Universal Robots URScript: infinity_multi.urscript

# UR10 -- infinity_multi
# Points: 3200   v=2.0 rad/s   a=1.7 rad/s2
# Generated by send_xyz.py
def run_infinity_multi():
  set_tool_voltage(12)           # power tool connector (12V for LED)
  set_tool_digital_out(0, False) # LED off initially
  movej([1.57, -1.2, 1.6, -0.4, 1.57, 0.0], a=0.4, v=0.2)   # go to home first
  movej([2.38, -1.326, 1.6, -0.4, 1.57, 0.0], a=0.4, v=0.2)   # move to pattern start
  sleep(1.5)   # pause — home ≠ start (dist=0.820 rad)
  set_tool_digital_out(0, True)  # LED on — drawing starts
  movej([2.38, -1.3359, 1.6, -0.4, 1.57, 0.0], a=1.7, v=2.0, r=0.08)
  movej([2.3799, -1.3458, 1.6, -0.4, 1.57, 0.0], a=1.7, v=2.0, r=0.08)
  movej([2.3798, -1.3557, 1.6, -0.4, 1.57, 0.0], a=1.7, v=2.0, r=0.08)
  movej([2.3796, -1.3656, 1.6, -0.4, 1.57, 0.0], a=1.7, v=2.0, r=0.08)
  movej([2.3794, -1.3755, 1.6, -0.4, 1.57, 0.0], a=1.7, v=2.0, r=0.08)
  movej([2.3791, -1.3854, 1.6, -0.4, 1.57, 0.0], a=1.7, v=2.0, r=0.08)
  movej([2.3788, -1.3952, 1.6, -0.4, 1.57, 0.0], a=1.7, v=2.0, r=0.08)
  movej([2.3784, -1.4051, 1.6, -0.4, 1.57, 0.0], a=1.7, v=2.0, r=0.08)
  movej([2.378, -1.4149, 1.6, -0.4, 1.57, 0.0], a=1.7, v=2.0, r=0.08)
  movej([2.3775, -1.4247, 1.6, -0.4, 1.57, 0.0], a=1.7, v=2.0, r=0.08)
  movej([2.377, -1.4344, 1.6, -0.4, 1.57, 0.0], a=1.7, v=2.0, r=0.08)
  movej([2.3764, -1.4442, 1.6, -0.4, 1.57, 0.0], a=1.7, v=2.0, r=0.08)
  movej([2.3758, -1.4539, 1.6, -0.4, 1.57, 0.0], a=1.7, v=2.0, r=0.08)
  movej([2.3751, -1.4636, 1.6, -0.4, 1.57, 0.0], a=1.7, v=2.0, r=0.08)
  movej([2.3744, -1.4733, 1.6, -0.4, 1.57, 0.0], a=1.7, v=2.0, r=0.08)
  movej([2.3736, -1.4829, 1.6, -0.4, 1.57, 0.0], a=1.7, v=2.0, r=0.08)
  movej([2.3728, -1.4924, 1.6, -0.4, 1.57, 0.0], a=1.7, v=2.0, r=0.08)
  movej([2.3719, -1.502, 1.6, -0.4, 1.57, 0.0], a=1.7, v=2.0, r=0.08)
  movej([2.371, -1.5115, 1.6, -0.4, 1.57, 0.0], a=1.7, v=2.0, r=0.08)
  movej([2.37, -1.5209, 1.6, -0.4, 1.57, 0.0], a=1.7, v=2.0, r=0.08)
  movej([2.369, -1.5303, 1.6, -0.4, 1.57, 0.0], a=1.7, v=2.0, r=0.08)
  movej([2.3679, -1.5397, 1.6, -0.4, 1.57, 0.0], a=1.7, v=2.0, r=0.08)
  movej([2.3668, -1.549, 1.6, -0.4, 1.57, 0.0], a=1.7, v=2.0, r=0.08)
  movej([2.3656, -1.5582, 1.6, -0.4, 1.57, 0.0], a=1.7, v=2.0, r=0.08)
  movej([2.3644, -1.5674, 1.6, -0.4, 1.57, 0.0], a=1.7, v=2.0, r=0.08)
  movej([2.3631, -1.5765, 1.6, -0.4, 1.57, 0.0], a=1.7, v=2.0, r=0.08)
  movej([2.3618, -1.5856, 1.6, -0.4, 1.57, 0.0], a=1.7, v=2.0, r=0.08)
  movej([2.3604, -1.5946, 1.6, -0.4, 1.57, 0.0], a=1.7, v=2.0, r=0.08)
  movej([2.359, -1.6035, 1.6, -0.4, 1.57, 0.0], a=1.7, v=2.0, r=0.08)
  movej([2.3576, -1.6123, 1.6, -0.4, 1.57, 0.0], a=1.7, v=2.0, r=0.08)
  movej([2.3561, -1.6211, 1.6, -0.4, 1.57, 0.0], a=1.7, v=2.0, r=0.08)
  movej([2.3545, -1.6299, 1.6, -0.4, 1.57, 0.0], a=1.7, v=2.0, r=0.08)
  movej([2.3529, -1.6385, 1.6, -0.4, 1.57, 0.0], a=1.7, v=2.0, r=0.08)
  movej([2.3512, -1.6471, 1.6, -0.4, 1.57, 0.0], a=1.7, v=2.0, r=0.08)
  movej([2.3495, -1.6555, 1.6, -0.4, 1.57, 0.0], a=1.7, v=2.0, r=0.08)
  movej([2.3478, -1.6639, 1.6, -0.4, 1.57, 0.0], a=1.7, v=2.0, r=0.08)
  movej([2.346, -1.6723, 1.6, -0.4, 1.57, 0.0], a=1.7, v=2.0, r=0.08)
  movej([2.3441, -1.6805, 1.6, -0.4, 1.57, 0.0], a=1.7, v=2.0, r=0.08)
  movej([2.3422, -1.6886, 1.6, -0.4, 1.57, 0.0], a=1.7, v=2.0, r=0.08)
  movej([2.3403, -1.6967, 1.6, -0.4, 1.57, 0.0], a=1.7, v=2.0, r=0.08)
  movej([2.3383, -1.7047, 1.6, -0.4, 1.57, 0.0], a=1.7, v=2.0, r=0.08)
  movej([2.3362, -1.7125, 1.6, -0.4, 1.57, 0.0], a=1.7, v=2.0, r=0.08)
  movej([2.3341, -1.7203, 1.6, -0.4, 1.57, 0.0], a=1.7, v=2.0, r=0.08)
  movej([2.332, -1.728, 1.6, -0.4, 1.57, 0.0], a=1.7, v=2.0, r=0.08)
  movej([2.3298, -1.7356, 1.6, -0.4, 1.57, 0.0], a=1.7, v=2.0, r=0.08)
  movej([2.3276, -1.7431, 1.6, -0.4, 1.57, 0.0], a=1.7, v=2.0, r=0.08)
  movej([2.3253, -1.7504, 1.6, -0.4, 1.57, 0.0], a=1.7, v=2.0, r=0.08)
  movej([2.323, -1.7577, 1.6, -0.4, 1.57, 0.0], a=1.7, v=2.0, r=0.08)
  movej([2.3206, -1.7649, 1.6, -0.4, 1.57, 0.0], a=1.7, v=2.0, r=0.08)
  movej([2.3182, -1.7719, 1.6, -0.4, 1.57, 0.0], a=1.7, v=2.0, r=0.08)
  movej([2.3157, -1.7789, 1.6, -0.4, 1.57, 0.0], a=1.7, v=2.0, r=0.08)
  movej([2.3132, -1.7857, 1.6, -0.4, 1.57, 0.0], a=1.7, v=2.0, r=0.08)
  movej([2.3107, -1.7924, 1.6, -0.4, 1.57, 0.0], a=1.7, v=2.0, r=0.08)
  movej([2.3081, -1.799, 1.6, -0.4, 1.57, 0.0], a=1.7, v=2.0, r=0.08)
  movej([2.3054, -1.8055, 1.6, -0.4, 1.57, 0.0], a=1.7, v=2.0, r=0.08)
  movej([2.3027, -1.8119, 1.6, -0.4, 1.57, 0.0], a=1.7, v=2.0, r=0.08)
  movej([2.3, -1.8181, 1.6, -0.4, 1.57, 0.0], a=1.7, v=2.0, r=0.08)
  movej([2.2972, -1.8242, 1.6, -0.4, 1.57, 0.0], a=1.7, v=2.0, r=0.08)
  movej([2.2944, -1.8302, 1.6, -0.4, 1.57, 0.0], a=1.7, v=2.0, r=0.08)
  movej([2.2915, -1.8361, 1.6, -0.4, 1.57, 0.0], a=1.7, v=2.0, r=0.08)
  movej([2.2886, -1.8419, 1.6, -0.4, 1.57, 0.0], a=1.7, v=2.0, r=0.08)
  movej([2.2856, -1.8475, 1.6, -0.4, 1.57, 0.0], a=1.7, v=2.0, r=0.08)
  movej([2.2826, -1.853, 1.6, -0.4, 1.57, 0.0], a=1.7, v=2.0, r=0.08)
  movej([2.2796, -1.8584, 1.6, -0.4, 1.57, 0.0], a=1.7, v=2.0, r=0.08)
  movej([2.2765, -1.8636, 1.6, -0.4, 1.57, 0.0], a=1.7, v=2.0, r=0.08)
  movej([2.2733, -1.8687, 1.6, -0.4, 1.57, 0.0], a=1.7, v=2.0, r=0.08)
  movej([2.2701, -1.8736, 1.6, -0.4, 1.57, 0.0], a=1.7, v=2.0, r=0.08)
  movej([2.2669, -1.8785, 1.6, -0.4, 1.57, 0.0], a=1.7, v=2.0, r=0.08)
  movej([2.2637, -1.8832, 1.6, -0.4, 1.57, 0.0], a=1.7, v=2.0, r=0.08)
  movej([2.2603, -1.8877, 1.6, -0.4, 1.57, 0.0], a=1.7, v=2.0, r=0.08)
  movej([2.257, -1.8921, 1.6, -0.4, 1.57, 0.0], a=1.7, v=2.0, r=0.08)
  movej([2.2536, -1.8964, 1.6, -0.4, 1.57, 0.0], a=1.7, v=2.0, r=0.08)
  movej([2.2502, -1.9006, 1.6, -0.4, 1.57, 0.0], a=1.7, v=2.0, r=0.08)
  movej([2.2467, -1.9045, 1.6, -0.4, 1.57, 0.0], a=1.7, v=2.0, r=0.08)
  movej([2.2432, -1.9084, 1.6, -0.4, 1.57, 0.0], a=1.7, v=2.0, r=0.08)
  movej([2.2396, -1.9121, 1.6, -0.4, 1.57, 0.0], a=1.7, v=2.0, r=0.08)
  movej([2.236, -1.9157, 1.6, -0.4, 1.57, 0.0], a=1.7, v=2.0, r=0.08)
  movej([2.2323, -1.9191, 1.6, -0.4, 1.57, 0.0], a=1.7, v=2.0, r=0.08)
  movej([2.2287, -1.9224, 1.6, -0.4, 1.57, 0.0], a=1.7, v=2.0, r=0.08)
  movej([2.2249, -1.9255, 1.6, -0.4, 1.57, 0.0], a=1.7, v=2.0, r=0.08)
  movej([2.2212, -1.9284, 1.6, -0.4, 1.57, 0.0], a=1.7, v=2.0, r=0.08)
  movej([2.2174, -1.9313, 1.6, -0.4, 1.57, 0.0], a=1.7, v=2.0, r=0.08)
  movej([2.2135, -1.9339, 1.6, -0.4, 1.57, 0.0], a=1.7, v=2.0, r=0.08)
  movej([2.2096, -1.9365, 1.6, -0.4, 1.57, 0.0], a=1.7, v=2.0, r=0.08)
  movej([2.2057, -1.9388, 1.6, -0.4, 1.57, 0.0], a=1.7, v=2.0, r=0.08)
  movej([2.2017, -1.9411, 1.6, -0.4, 1.57, 0.0], a=1.7, v=2.0, r=0.08)
  movej([2.1977, -1.9431, 1.6, -0.4, 1.57, 0.0], a=1.7, v=2.0, r=0.08)
  movej([2.1937, -1.945, 1.6, -0.4, 1.57, 0.0], a=1.7, v=2.0, r=0.08)
  movej([2.1896, -1.9468, 1.6, -0.4, 1.57, 0.0], a=1.7, v=2.0, r=0.08)
  movej([2.1855, -1.9484, 1.6, -0.4, 1.57, 0.0], a=1.7, v=2.0, r=0.08)
  movej([2.1813, -1.9499, 1.6, -0.4, 1.57, 0.0], a=1.7, v=2.0, r=0.08)
  movej([2.1771, -1.9512, 1.6, -0.4, 1.57, 0.0], a=1.7, v=2.0, r=0.08)
  movej([2.1729, -1.9523, 1.6, -0.4, 1.57, 0.0], a=1.7, v=2.0, r=0.08)
  movej([2.1686, -1.9533, 1.6, -0.4, 1.57, 0.0], a=1.7, v=2.0, r=0.08)
  movej([2.1643, -1.9542, 1.6, -0.4, 1.57, 0.0], a=1.7, v=2.0, r=0.08)
  movej([2.1599, -1.9548, 1.6, -0.4, 1.57, 0.0], a=1.7, v=2.0, r=0.08)
  movej([2.1556, -1.9554, 1.6, -0.4, 1.57, 0.0], a=1.7, v=2.0, r=0.08)
  movej([2.1511, -1.9557, 1.6, -0.4, 1.57, 0.0], a=1.7, v=2.0, r=0.08)
  movej([2.1467, -1.9559, 1.6, -0.4, 1.57, 0.0], a=1.7, v=2.0, r=0.08)
  movej([2.1422, -1.956, 1.6, -0.4, 1.57, 0.0], a=1.7, v=2.0, r=0.08)
  movej([2.1377, -1.9559, 1.6, -0.4, 1.57, 0.0], a=1.7, v=2.0, r=0.08)
  movej([2.1331, -1.9556, 1.6, -0.4, 1.57, 0.0], a=1.7, v=2.0, r=0.08)
  movej([2.1285, -1.9552, 1.6, -0.4, 1.57, 0.0], a=1.7, v=2.0, r=0.08)
  movej([2.1239, -1.9547, 1.6, -0.4, 1.57, 0.0], a=1.7, v=2.0, r=0.08)
  movej([2.1192, -1.954, 1.6, -0.4, 1.57, 0.0], a=1.7, v=2.0, r=0.08)
  movej([2.1145, -1.9531, 1.6, -0.4, 1.57, 0.0], a=1.7, v=2.0, r=0.08)
  movej([2.1098, -1.952, 1.6, -0.4, 1.57, 0.0], a=1.7, v=2.0, r=0.08)
  movej([2.105, -1.9509, 1.6, -0.4, 1.57, 0.0], a=1.7, v=2.0, r=0.08)
  movej([2.1002, -1.9495, 1.6, -0.4, 1.57, 0.0], a=1.7, v=2.0, r=0.08)
  movej([2.0954, -1.948, 1.6, -0.4, 1.57, 0.0], a=1.7, v=2.0, r=0.08)
  movej([2.0905, -1.9464, 1.6, -0.4, 1.57, 0.0], a=1.7, v=2.0, r=0.08)
  movej([2.0856, -1.9446, 1.6, -0.4, 1.57, 0.0], a=1.7, v=2.0, r=0.08)
  movej([2.0807, -1.9426, 1.6, -0.4, 1.57, 0.0], a=1.7, v=2.0, r=0.08)
  movej([2.0757, -1.9405, 1.6, -0.4, 1.57, 0.0], a=1.7, v=2.0, r=0.08)
  movej([2.0707, -1.9383, 1.6, -0.4, 1.57, 0.0], a=1.7, v=2.0, r=0.08)
  movej([2.0657, -1.9358, 1.6, -0.4, 1.57, 0.0], a=1.7, v=2.0, r=0.08)
  movej([2.0607, -1.9333, 1.6, -0.4, 1.57, 0.0], a=1.7, v=2.0, r=0.08)
  movej([2.0556, -1.9306, 1.6, -0.4, 1.57, 0.0], a=1.7, v=2.0, r=0.08)
  movej([2.0505, -1.9277, 1.6, -0.4, 1.57, 0.0], a=1.7, v=2.0, r=0.08)
  movej([2.0453, -1.9247, 1.6, -0.4, 1.57, 0.0], a=1.7, v=2.0, r=0.08)
  movej([2.0402, -1.9215, 1.6, -0.4, 1.57, 0.0], a=1.7, v=2.0, r=0.08)
  movej([2.035, -1.9182, 1.6, -0.4, 1.57, 0.0], a=1.7, v=2.0, r=0.08)
  movej([2.0297, -1.9148, 1.6, -0.4, 1.57, 0.0], a=1.7, v=2.0, r=0.08)
  movej([2.0245, -1.9112, 1.6, -0.4, 1.57, 0.0], a=1.7, v=2.0, r=0.08)
  movej([2.0192, -1.9075, 1.6, -0.4, 1.57, 0.0], a=1.7, v=2.0, r=0.08)
  movej([2.0139, -1.9036, 1.6, -0.4, 1.57, 0.0], a=1.7, v=2.0, r=0.08)
  movej([2.0085, -1.8995, 1.6, -0.4, 1.57, 0.0], a=1.7, v=2.0, r=0.08)
  movej([2.0032, -1.8954, 1.6, -0.4, 1.57, 0.0], a=1.7, v=2.0, r=0.08)
  movej([1.9978, -1.8911, 1.6, -0.4, 1.57, 0.0], a=1.7, v=2.0, r=0.08)
  movej([1.9923, -1.8866, 1.6, -0.4, 1.57, 0.0], a=1.7, v=2.0, r=0.08)
  movej([1.9869, -1.882, 1.6, -0.4, 1.57, 0.0], a=1.7, v=2.0, r=0.08)
  movej([1.9814, -1.8773, 1.6, -0.4, 1.57, 0.0], a=1.7, v=2.0, r=0.08)
  movej([1.9759, -1.8724, 1.6, -0.4, 1.57, 0.0], a=1.7, v=2.0, r=0.08)
  movej([1.9704, -1.8674, 1.6, -0.4, 1.57, 0.0], a=1.7, v=2.0, r=0.08)
  movej([1.9648, -1.8623, 1.6, -0.4, 1.57, 0.0], a=1.7, v=2.0, r=0.08)
  movej([1.9593, -1.857, 1.6, -0.4, 1.57, 0.0], a=1.7, v=2.0, r=0.08)
  movej([1.9537, -1.8516, 1.6, -0.4, 1.57, 0.0], a=1.7, v=2.0, r=0.08)
  movej([1.9481, -1.8461, 1.6, -0.4, 1.57, 0.0], a=1.7, v=2.0, r=0.08)
  movej([1.9424, -1.8404, 1.6, -0.4, 1.57, 0.0], a=1.7, v=2.0, r=0.08)
  movej([1.9367, -1.8347, 1.6, -0.4, 1.57, 0.0], a=1.7, v=2.0, r=0.08)
  movej([1.931, -1.8288, 1.6, -0.4, 1.57, 0.0], a=1.7, v=2.0, r=0.08)
  movej([1.9253, -1.8227, 1.6, -0.4, 1.57, 0.0], a=1.7, v=2.0, r=0.08)
  movej([1.9196, -1.8166, 1.6, -0.4, 1.57, 0.0], a=1.7, v=2.0, r=0.08)
  movej([1.9138, -1.8103, 1.6, -0.4, 1.57, 0.0], a=1.7, v=2.0, r=0.08)
  movej([1.9081, -1.8039, 1.6, -0.4, 1.57, 0.0], a=1.7, v=2.0, r=0.08)
  movej([1.9023, -1.7974, 1.6, -0.4, 1.57, 0.0], a=1.7, v=2.0, r=0.08)
  movej([1.8964, -1.7907, 1.6, -0.4, 1.57, 0.0], a=1.7, v=2.0, r=0.08)
  movej([1.8906, -1.784, 1.6, -0.4, 1.57, 0.0], a=1.7, v=2.0, r=0.08)
  movej([1.8847, -1.7771, 1.6, -0.4, 1.57, 0.0], a=1.7, v=2.0, r=0.08)
  movej([1.8789, -1.7702, 1.6, -0.4, 1.57, 0.0], a=1.7, v=2.0, r=0.08)
  movej([1.873, -1.7631, 1.6, -0.4, 1.57, 0.0], a=1.7, v=2.0, r=0.08)
  movej([1.8671, -1.7559, 1.6, -0.4, 1.57, 0.0], a=1.7, v=2.0, r=0.08)
  movej([1.8611, -1.7486, 1.6, -0.4, 1.57, 0.0], a=1.7, v=2.0, r=0.08)
  movej([1.8552, -1.7412, 1.6, -0.4, 1.57, 0.0], a=1.7, v=2.0, r=0.08)
  movej([1.8492, -1.7337, 1.6, -0.4, 1.57, 0.0], a=1.7, v=2.0, r=0.08)
  movej([1.8432, -1.7261, 1.6, -0.4, 1.57, 0.0], a=1.7, v=2.0, r=0.08)
  movej([1.8372, -1.7184, 1.6, -0.4, 1.57, 0.0], a=1.7, v=2.0, r=0.08)
  movej([1.8312, -1.7106, 1.6, -0.4, 1.57, 0.0], a=1.7, v=2.0, r=0.08)
  movej([1.8251, -1.7027, 1.6, -0.4, 1.57, 0.0], a=1.7, v=2.0, r=0.08)
  movej([1.8191, -1.6947, 1.6, -0.4, 1.57, 0.0], a=1.7, v=2.0, r=0.08)
  movej([1.813, -1.6866, 1.6, -0.4, 1.57, 0.0], a=1.7, v=2.0, r=0.08)
  movej([1.8069, -1.6785, 1.6, -0.4, 1.57, 0.0], a=1.7, v=2.0, r=0.08)
  movej([1.8008, -1.6702, 1.6, -0.4, 1.57, 0.0], a=1.7, v=2.0, r=0.08)
  movej([1.7947, -1.6619, 1.6, -0.4, 1.57, 0.0], a=1.7, v=2.0, r=0.08)
  movej([1.7886, -1.6534, 1.6, -0.4, 1.57, 0.0], a=1.7, v=2.0, r=0.08)
  movej([1.7825, -1.6449, 1.6, -0.4, 1.57, 0.0], a=1.7, v=2.0, r=0.08)
  movej([1.7763, -1.6363, 1.6, -0.4, 1.57, 0.0], a=1.7, v=2.0, r=0.08)
  movej([1.7701, -1.6277, 1.6, -0.4, 1.57, 0.0], a=1.7, v=2.0, r=0.08)
  movej([1.764, -1.6189, 1.6, -0.4, 1.57, 0.0], a=1.7, v=2.0, r=0.08)
  movej([1.7578, -1.6101, 1.6, -0.4, 1.57, 0.0], a=1.7, v=2.0, r=0.08)
  movej([1.7516, -1.6013, 1.6, -0.4, 1.57, 0.0], a=1.7, v=2.0, r=0.08)
  movej([1.7454, -1.5923, 1.6, -0.4, 1.57, 0.0], a=1.7, v=2.0, r=0.08)
  movej([1.7391, -1.5833, 1.6, -0.4, 1.57, 0.0], a=1.7, v=2.0, r=0.08)
  movej([1.7329, -1.5742, 1.6, -0.4, 1.57, 0.0], a=1.7, v=2.0, r=0.08)
  movej([1.7267, -1.5651, 1.6, -0.4, 1.57, 0.0], a=1.7, v=2.0, r=0.08)
  movej([1.7204, -1.5559, 1.6, -0.4, 1.57, 0.0], a=1.7, v=2.0, r=0.08)
  movej([1.7141, -1.5466, 1.6, -0.4, 1.57, 0.0], a=1.7, v=2.0, r=0.08)
  movej([1.7079, -1.5373, 1.6, -0.4, 1.57, 0.0], a=1.7, v=2.0, r=0.08)
  movej([1.7016, -1.528, 1.6, -0.4, 1.57, 0.0], a=1.7, v=2.0, r=0.08)
  movej([1.6953, -1.5186, 1.6, -0.4, 1.57, 0.0], a=1.7, v=2.0, r=0.08)
  movej([1.689, -1.5091, 1.6, -0.4, 1.57, 0.0], a=1.7, v=2.0, r=0.08)
  movej([1.6827, -1.4996, 1.6, -0.4, 1.57, 0.0], a=1.7, v=2.0, r=0.08)
  movej([1.6764, -1.4901, 1.6, -0.4, 1.57, 0.0], a=1.7, v=2.0, r=0.08)
  movej([1.6701, -1.4805, 1.6, -0.4, 1.57, 0.0], a=1.7, v=2.0, r=0.08)
  movej([1.6637, -1.4708, 1.6, -0.4, 1.57, 0.0], a=1.7, v=2.0, r=0.08)
  movej([1.6574, -1.4612, 1.6, -0.4, 1.57, 0.0], a=1.7, v=2.0, r=0.08)
  movej([1.6511, -1.4515, 1.6, -0.4, 1.57, 0.0], a=1.7, v=2.0, r=0.08)
  movej([1.6447, -1.4418, 1.6, -0.4, 1.57, 0.0], a=1.7, v=2.0, r=0.08)
  movej([1.6384, -1.432, 1.6, -0.4, 1.57, 0.0], a=1.7, v=2.0, r=0.08)
  movej([1.632, -1.4222, 1.6, -0.4, 1.57, 0.0], a=1.7, v=2.0, r=0.08)
  movej([1.6257, -1.4124, 1.6, -0.4, 1.57, 0.0], a=1.7, v=2.0, r=0.08)
  movej([1.6193, -1.4026, 1.6, -0.4, 1.57, 0.0], a=1.7, v=2.0, r=0.08)
  movej([1.613, -1.3928, 1.6, -0.4, 1.57, 0.0], a=1.7, v=2.0, r=0.08)
  movej([1.6066, -1.3829, 1.6, -0.4, 1.57, 0.0], a=1.7, v=2.0, r=0.08)
  movej([1.6002, -1.373, 1.6, -0.4, 1.57, 0.0], a=1.7, v=2.0, r=0.08)
  movej([1.5939, -1.3631, 1.6, -0.4, 1.57, 0.0], a=1.7, v=2.0, r=0.08)
  movej([1.5875, -1.3532, 1.6, -0.4, 1.57, 0.0], a=1.7, v=2.0, r=0.08)
  movej([1.5811, -1.3433, 1.6, -0.4, 1.57, 0.0], a=1.7, v=2.0, r=0.08)
  movej([1.5748, -1.3334, 1.6, -0.4, 1.57, 0.0], a=1.7, v=2.0, r=0.08)
  movej([1.5684, -1.3235, 1.6, -0.4, 1.57, 0.0], a=1.7, v=2.0, r=0.08)
  movej([1.562, -1.3136, 1.6, -0.4, 1.57, 0.0], a=1.7, v=2.0, r=0.08)
  movej([1.5557, -1.3037, 1.6, -0.4, 1.57, 0.0], a=1.7, v=2.0, r=0.08)
  movej([1.5493, -1.2938, 1.6, -0.4, 1.57, 0.0], a=1.7, v=2.0, r=0.08)
  movej([1.5429, -1.2839, 1.6, -0.4, 1.57, 0.0], a=1.7, v=2.0, r=0.08)
  movej([1.5366, -1.274, 1.6, -0.4, 1.57, 0.0], a=1.7, v=2.0, r=0.08)
  movej([1.5302, -1.2642, 1.6, -0.4, 1.57, 0.0], a=1.7, v=2.0, r=0.08)
  movej([1.5238, -1.2543, 1.6, -0.4, 1.57, 0.0], a=1.7, v=2.0, r=0.08)
  movej([1.5175, -1.2445, 1.6, -0.4, 1.57, 0.0], a=1.7, v=2.0, r=0.08)
  movej([1.5111, -1.2347, 1.6, -0.4, 1.57, 0.0], a=1.7, v=2.0, r=0.08)
  movej([1.5048, -1.2249, 1.6, -0.4, 1.57, 0.0], a=1.7, v=2.0, r=0.08)
  movej([1.4984, -1.2151, 1.6, -0.4, 1.57, 0.0], a=1.7, v=2.0, r=0.08)
  movej([1.4921, -1.2054, 1.6, -0.4, 1.57, 0.0], a=1.7, v=2.0, r=0.08)
  movej([1.4858, -1.1957, 1.6, -0.4, 1.57, 0.0], a=1.7, v=2.0, r=0.08)
  movej([1.4794, -1.186, 1.6, -0.4, 1.57, 0.0], a=1.7, v=2.0, r=0.08)
  movej([1.4731, -1.1763, 1.6, -0.4, 1.57, 0.0], a=1.7, v=2.0, r=0.08)
  movej([1.4668, -1.1667, 1.6, -0.4, 1.57, 0.0], a=1.7, v=2.0, r=0.08)
  movej([1.4605, -1.1572, 1.6, -0.4, 1.57, 0.0], a=1.7, v=2.0, r=0.08)
  movej([1.4541, -1.1476, 1.6, -0.4, 1.57, 0.0], a=1.7, v=2.0, r=0.08)
  movej([1.4478, -1.1382, 1.6, -0.4, 1.57, 0.0], a=1.7, v=2.0, r=0.08)
  movej([1.4416, -1.1287, 1.6, -0.4, 1.57, 0.0], a=1.7, v=2.0, r=0.08)
  movej([1.4353, -1.1193, 1.6, -0.4, 1.57, 0.0], a=1.7, v=2.0, r=0.08)
  movej([1.429, -1.11, 1.6, -0.4, 1.57, 0.0], a=1.7, v=2.0, r=0.08)
  movej([1.4227, -1.1007, 1.6, -0.4, 1.57, 0.0], a=1.7, v=2.0, r=0.08)
  movej([1.4165, -1.0915, 1.6, -0.4, 1.57, 0.0], a=1.7, v=2.0, r=0.08)
  movej([1.4102, -1.0823, 1.6, -0.4, 1.57, 0.0], a=1.7, v=2.0, r=0.08)
  movej([1.404, -1.0732, 1.6, -0.4, 1.57, 0.0], a=1.7, v=2.0, r=0.08)
  movej([1.3977, -1.0642, 1.6, -0.4, 1.57, 0.0], a=1.7, v=2.0, r=0.08)
  movej([1.3915, -1.0552, 1.6, -0.4, 1.57, 0.0], a=1.7, v=2.0, r=0.08)
  movej([1.3853, -1.0463, 1.6, -0.4, 1.57, 0.0], a=1.7, v=2.0, r=0.08)
  movej([1.3791, -1.0375, 1.6, -0.4, 1.57, 0.0], a=1.7, v=2.0, r=0.08)
  movej([1.3729, -1.0287, 1.6, -0.4, 1.57, 0.0], a=1.7, v=2.0, r=0.08)
  movej([1.3668, -1.02, 1.6, -0.4, 1.57, 0.0], a=1.7, v=2.0, r=0.08)
  movej([1.3606, -1.0114, 1.6, -0.4, 1.57, 0.0], a=1.7, v=2.0, r=0.08)
  movej([1.3545, -1.0028, 1.6, -0.4, 1.57, 0.0], a=1.7, v=2.0, r=0.08)
  movej([1.3483, -0.9943, 1.6, -0.4, 1.57, 0.0], a=1.7, v=2.0, r=0.08)
  movej([1.3422, -0.986, 1.6, -0.4, 1.57, 0.0], a=1.7, v=2.0, r=0.08)
  movej([1.3361, -0.9777, 1.6, -0.4, 1.57, 0.0], a=1.7, v=2.0, r=0.08)
  movej([1.33, -0.9695, 1.6, -0.4, 1.57, 0.0], a=1.7, v=2.0, r=0.08)
  movej([1.3239, -0.9613, 1.6, -0.4, 1.57, 0.0], a=1.7, v=2.0, r=0.08)
  movej([1.3179, -0.9533, 1.6, -0.4, 1.57, 0.0], a=1.7, v=2.0, r=0.08)
  movej([1.3118, -0.9454, 1.6, -0.4, 1.57, 0.0], a=1.7, v=2.0, r=0.08)
  movej([1.3058, -0.9375, 1.6, -0.4, 1.57, 0.0], a=1.7, v=2.0, r=0.08)
  movej([1.2998, -0.9298, 1.6, -0.4, 1.57, 0.0], a=1.7, v=2.0, r=0.08)
  movej([1.2938, -0.9221, 1.6, -0.4, 1.57, 0.0], a=1.7, v=2.0, r=0.08)
  movej([1.2878, -0.9145, 1.6, -0.4, 1.57, 0.0], a=1.7, v=2.0, r=0.08)
  movej([1.2818, -0.9071, 1.6, -0.4, 1.57, 0.0], a=1.7, v=2.0, r=0.08)
  movej([1.2759, -0.8997, 1.6, -0.4, 1.57, 0.0], a=1.7, v=2.0, r=0.08)
  movej([1.27, -0.8925, 1.6, -0.4, 1.57, 0.0], a=1.7, v=2.0, r=0.08)
  movej([1.2641, -0.8854, 1.6, -0.4, 1.57, 0.0], a=1.7, v=2.0, r=0.08)
  movej([1.2582, -0.8783, 1.6, -0.4, 1.57, 0.0], a=1.7, v=2.0, r=0.08)
  movej([1.2523, -0.8714, 1.6, -0.4, 1.57, 0.0], a=1.7, v=2.0, r=0.08)
  movej([1.2465, -0.8646, 1.6, -0.4, 1.57, 0.0], a=1.7, v=2.0, r=0.08)
  movej([1.2406, -0.8579, 1.6, -0.4, 1.57, 0.0], a=1.7, v=2.0, r=0.08)
  movej([1.2348, -0.8514, 1.6, -0.4, 1.57, 0.0], a=1.7, v=2.0, r=0.08)
  movej([1.229, -0.8449, 1.6, -0.4, 1.57, 0.0], a=1.7, v=2.0, r=0.08)
  movej([1.2233, -0.8386, 1.6, -0.4, 1.57, 0.0], a=1.7, v=2.0, r=0.08)
  movej([1.2175, -0.8323, 1.6, -0.4, 1.57, 0.0], a=1.7, v=2.0, r=0.08)
  movej([1.2118, -0.8262, 1.6, -0.4, 1.57, 0.0], a=1.7, v=2.0, r=0.08)
  movej([1.2061, -0.8203, 1.6, -0.4, 1.57, 0.0], a=1.7, v=2.0, r=0.08)
  movej([1.2004, -0.8144, 1.6, -0.4, 1.57, 0.0], a=1.7, v=2.0, r=0.08)
  movej([1.1948, -0.8087, 1.6, -0.4, 1.57, 0.0], a=1.7, v=2.0, r=0.08)
  movej([1.1891, -0.8031, 1.6, -0.4, 1.57, 0.0], a=1.7, v=2.0, r=0.08)
  movej([1.1835, -0.7977, 1.6, -0.4, 1.57, 0.0], a=1.7, v=2.0, r=0.08)
  movej([1.1779, -0.7923, 1.6, -0.4, 1.57, 0.0], a=1.7, v=2.0, r=0.08)
  movej([1.1724, -0.7871, 1.6, -0.4, 1.57, 0.0], a=1.7, v=2.0, r=0.08)
  movej([1.1668, -0.7821, 1.6, -0.4, 1.57, 0.0], a=1.7, v=2.0, r=0.08)
  movej([1.1613, -0.7771, 1.6, -0.4, 1.57, 0.0], a=1.7, v=2.0, r=0.08)
  movej([1.1558, -0.7723, 1.6, -0.4, 1.57, 0.0], a=1.7, v=2.0, r=0.08)
  movej([1.1504, -0.7677, 1.6, -0.4, 1.57, 0.0], a=1.7, v=2.0, r=0.08)
  movej([1.1449, -0.7632, 1.6, -0.4, 1.57, 0.0], a=1.7, v=2.0, r=0.08)
  movej([1.1395, -0.7588, 1.6, -0.4, 1.57, 0.0], a=1.7, v=2.0, r=0.08)
  movej([1.1341, -0.7545, 1.6, -0.4, 1.57, 0.0], a=1.7, v=2.0, r=0.08)
  movej([1.1288, -0.7504, 1.6, -0.4, 1.57, 0.0], a=1.7, v=2.0, r=0.08)
  movej([1.1235, -0.7465, 1.6, -0.4, 1.57, 0.0], a=1.7, v=2.0, r=0.08)
  movej([1.1182, -0.7427, 1.6, -0.4, 1.57, 0.0], a=1.7, v=2.0, r=0.08)
  movej([1.1129, -0.739, 1.6, -0.4, 1.57, 0.0], a=1.7, v=2.0, r=0.08)
  movej([1.1076, -0.7355, 1.6, -0.4, 1.57, 0.0], a=1.7, v=2.0, r=0.08)
  movej([1.1024, -0.7321, 1.6, -0.4, 1.57, 0.0], a=1.7, v=2.0, r=0.08)
  movej([1.0972, -0.7289, 1.6, -0.4, 1.57, 0.0], a=1.7, v=2.0, r=0.08)
  movej([1.0921, -0.7258, 1.6, -0.4, 1.57, 0.0], a=1.7, v=2.0, r=0.08)
  movej([1.087, -0.7228, 1.6, -0.4, 1.57, 0.0], a=1.7, v=2.0, r=0.08)
  movej([1.0819, -0.72, 1.6, -0.4, 1.57, 0.0], a=1.7, v=2.0, r=0.08)
  movej([1.0768, -0.7174, 1.6, -0.4, 1.57, 0.0], a=1.7, v=2.0, r=0.08)
  movej([1.0718, -0.7149, 1.6, -0.4, 1.57, 0.0], a=1.7, v=2.0, r=0.08)
  movej([1.0667, -0.7126, 1.6, -0.4, 1.57, 0.0], a=1.7, v=2.0, r=0.08)
  movej([1.0618, -0.7104, 1.6, -0.4, 1.57, 0.0], a=1.7, v=2.0, r=0.08)
  movej([1.0568, -0.7084, 1.6, -0.4, 1.57, 0.0], a=1.7, v=2.0, r=0.08)
  movej([1.0519, -0.7065, 1.6, -0.4, 1.57, 0.0], a=1.7, v=2.0, r=0.08)
  movej([1.047, -0.7048, 1.6, -0.4, 1.57, 0.0], a=1.7, v=2.0, r=0.08)
  movej([1.0422, -0.7032, 1.6, -0.4, 1.57, 0.0], a=1.7, v=2.0, r=0.08)
  movej([1.0374, -0.7018, 1.6, -0.4, 1.57, 0.0], a=1.7, v=2.0, r=0.08)
  movej([1.0326, -0.7005, 1.6, -0.4, 1.57, 0.0], a=1.7, v=2.0, r=0.08)
  movej([1.0278, -0.6994, 1.6, -0.4, 1.57, 0.0], a=1.7, v=2.0, r=0.08)
  movej([1.0231, -0.6985, 1.6, -0.4, 1.57, 0.0], a=1.7, v=2.0, r=0.08)
  movej([1.0184, -0.6977, 1.6, -0.4, 1.57, 0.0], a=1.7, v=2.0, r=0.08)
  movej([1.0138, -0.697, 1.6, -0.4, 1.57, 0.0], a=1.7, v=2.0, r=0.08)
  movej([1.0092, -0.6965, 1.6, -0.4, 1.57, 0.0], a=1.7, v=2.0, r=0.08)
  movej([1.0046, -0.6962, 1.6, -0.4, 1.57, 0.0], a=1.7, v=2.0, r=0.08)
  movej([1.0001, -0.696, 1.6, -0.4, 1.57, 0.0], a=1.7, v=2.0, r=0.08)
  movej([0.9956, -0.696, 1.6, -0.4, 1.57, 0.0], a=1.7, v=2.0, r=0.08)
  movej([0.9911, -0.6961, 1.6, -0.4, 1.57, 0.0], a=1.7, v=2.0, r=0.08)
  movej([0.9866, -0.6964, 1.6, -0.4, 1.57, 0.0], a=1.7, v=2.0, r=0.08)
  movej([0.9822, -0.6969, 1.6, -0.4, 1.57, 0.0], a=1.7, v=2.0, r=0.08)
  movej([0.9779, -0.6975, 1.6, -0.4, 1.57, 0.0], a=1.7, v=2.0, r=0.08)
  movej([0.9735, -0.6982, 1.6, -0.4, 1.57, 0.0], a=1.7, v=2.0, r=0.08)
  movej([0.9693, -0.6992, 1.6, -0.4, 1.57, 0.0], a=1.7, v=2.0, r=0.08)
  movej([0.965, -0.7002, 1.6, -0.4, 1.57, 0.0], a=1.7, v=2.0, r=0.08)
  movej([0.9608, -0.7015, 1.6, -0.4, 1.57, 0.0], a=1.7, v=2.0, r=0.08)
  movej([0.9566, -0.7028, 1.6, -0.4, 1.57, 0.0], a=1.7, v=2.0, r=0.08)
  movej([0.9525, -0.7044, 1.6, -0.4, 1.57, 0.0], a=1.7, v=2.0, r=0.08)
  movej([0.9484, -0.7061, 1.6, -0.4, 1.57, 0.0], a=1.7, v=2.0, r=0.08)
  movej([0.9443, -0.7079, 1.6, -0.4, 1.57, 0.0], a=1.7, v=2.0, r=0.08)
  movej([0.9403, -0.7099, 1.6, -0.4, 1.57, 0.0], a=1.7, v=2.0, r=0.08)
  movej([0.9363, -0.712, 1.6, -0.4, 1.57, 0.0], a=1.7, v=2.0, r=0.08)
  movej([0.9323, -0.7143, 1.6, -0.4, 1.57, 0.0], a=1.7, v=2.0, r=0.08)
  movej([0.9284, -0.7168, 1.6, -0.4, 1.57, 0.0], a=1.7, v=2.0, r=0.08)
  movej([0.9246, -0.7194, 1.6, -0.4, 1.57, 0.0], a=1.7, v=2.0, r=0.08)
  movej([0.9207, -0.7221, 1.6, -0.4, 1.57, 0.0], a=1.7, v=2.0, r=0.08)
  movej([0.9169, -0.725, 1.6, -0.4, 1.57, 0.0], a=1.7, v=2.0, r=0.08)
  movej([0.9132, -0.7281, 1.6, -0.4, 1.57, 0.0], a=1.7, v=2.0, r=0.08)
  movej([0.9095, -0.7313, 1.6, -0.4, 1.57, 0.0], a=1.7, v=2.0, r=0.08)
  movej([0.9058, -0.7346, 1.6, -0.4, 1.57, 0.0], a=1.7, v=2.0, r=0.08)
  movej([0.9022, -0.7381, 1.6, -0.4, 1.57, 0.0], a=1.7, v=2.0, r=0.08)
  movej([0.8986, -0.7417, 1.6, -0.4, 1.57, 0.0], a=1.7, v=2.0, r=0.08)
  movej([0.8951, -0.7455, 1.6, -0.4, 1.57, 0.0], a=1.7, v=2.0, r=0.08)
  movej([0.8916, -0.7494, 1.6, -0.4, 1.57, 0.0], a=1.7, v=2.0, r=0.08)
  movej([0.8881, -0.7535, 1.6, -0.4, 1.57, 0.0], a=1.7, v=2.0, r=0.08)
  movej([0.8847, -0.7577, 1.6, -0.4, 1.57, 0.0], a=1.7, v=2.0, r=0.08)
  movej([0.8813, -0.762, 1.6, -0.4, 1.57, 0.0], a=1.7, v=2.0, r=0.08)
  movej([0.878, -0.7665, 1.6, -0.4, 1.57, 0.0], a=1.7, v=2.0, r=0.08)
  movej([0.8747, -0.7712, 1.6, -0.4, 1.57, 0.0], a=1.7, v=2.0, r=0.08)
  movej([0.8715, -0.7759, 1.6, -0.4, 1.57, 0.0], a=1.7, v=2.0, r=0.08)
  movej([0.8682, -0.7808, 1.6, -0.4, 1.57, 0.0], a=1.7, v=2.0, r=0.08)
  movej([0.8651, -0.7858, 1.6, -0.4, 1.57, 0.0], a=1.7, v=2.0, r=0.08)
  movej([0.862, -0.791, 1.6, -0.4, 1.57, 0.0], a=1.7, v=2.0, r=0.08)
  movej([0.8589, -0.7963, 1.6, -0.4, 1.57, 0.0], a=1.7, v=2.0, r=0.08)
  movej([0.8559, -0.8017, 1.6, -0.4, 1.57, 0.0], a=1.7, v=2.0, r=0.08)
  movej([0.8529, -0.8073, 1.6, -0.4, 1.57, 0.0], a=1.7, v=2.0, r=0.08)
  movej([0.8499, -0.813, 1.6, -0.4, 1.57, 0.0], a=1.7, v=2.0, r=0.08)
  movej([0.8471, -0.8188, 1.6, -0.4, 1.57, 0.0], a=1.7, v=2.0, r=0.08)
  movej([0.8442, -0.8247, 1.6, -0.4, 1.57, 0.0], a=1.7, v=2.0, r=0.08)
  movej([0.8414, -0.8308, 1.6, -0.4, 1.57, 0.0], a=1.7, v=2.0, r=0.08)
  movej([0.8386, -0.837, 1.6, -0.4, 1.57, 0.0], a=1.7, v=2.0, r=0.08)
  movej([0.8359, -0.8433, 1.6, -0.4, 1.57, 0.0], a=1.7, v=2.0, r=0.08)
  movej([0.8333, -0.8497, 1.6, -0.4, 1.57, 0.0], a=1.7, v=2.0, r=0.08)
  movej([0.8306, -0.8563, 1.6, -0.4, 1.57, 0.0], a=1.7, v=2.0, r=0.08)
  movej([0.828, -0.8629, 1.6, -0.4, 1.57, 0.0], a=1.7, v=2.0, r=0.08)
  movej([0.8255, -0.8697, 1.6, -0.4, 1.57, 0.0], a=1.7, v=2.0, r=0.08)
  movej([0.823, -0.8766, 1.6, -0.4, 1.57, 0.0], a=1.7, v=2.0, r=0.08)
  movej([0.8206, -0.8836, 1.6, -0.4, 1.57, 0.0], a=1.7, v=2.0, r=0.08)
  movej([0.8182, -0.8907, 1.6, -0.4, 1.57, 0.0], a=1.7, v=2.0, r=0.08)
  movej([0.8158, -0.8979, 1.6, -0.4, 1.57, 0.0], a=1.7, v=2.0, r=0.08)
  movej([0.8135, -0.9052, 1.6, -0.4, 1.57, 0.0], a=1.7, v=2.0, r=0.08)
  movej([0.8113, -0.9127, 1.6, -0.4, 1.57, 0.0], a=1.7, v=2.0, r=0.08)
  movej([0.8091, -0.9202, 1.6, -0.4, 1.57, 0.0], a=1.7, v=2.0, r=0.08)
  movej([0.8069, -0.9278, 1.6, -0.4, 1.57, 0.0], a=1.7, v=2.0, r=0.08)
  movej([0.8048, -0.9356, 1.6, -0.4, 1.57, 0.0], a=1.7, v=2.0, r=0.08)
  movej([0.8027, -0.9434, 1.6, -0.4, 1.57, 0.0], a=1.7, v=2.0, r=0.08)
  movej([0.8007, -0.9513, 1.6, -0.4, 1.57, 0.0], a=1.7, v=2.0, r=0.08)
  movej([0.7988, -0.9593, 1.6, -0.4, 1.57, 0.0], a=1.7, v=2.0, r=0.08)
  movej([0.7968, -0.9674, 1.6, -0.4, 1.57, 0.0], a=1.7, v=2.0, r=0.08)
  movej([0.795, -0.9756, 1.6, -0.4, 1.57, 0.0], a=1.7, v=2.0, r=0.08)
  movej([0.7931, -0.9839, 1.6, -0.4, 1.57, 0.0], a=1.7, v=2.0, r=0.08)
  movej([0.7914, -0.9922, 1.6, -0.4, 1.57, 0.0], a=1.7, v=2.0, r=0.08)
  movej([0.7896, -1.0007, 1.6, -0.4, 1.57, 0.0], a=1.7, v=2.0, r=0.08)
  movej([0.7879, -1.0092, 1.6, -0.4, 1.57, 0.0], a=1.7, v=2.0, r=0.08)
  movej([0.7863, -1.0178, 1.6, -0.4, 1.57, 0.0], a=1.7, v=2.0, r=0.08)
  movej([0.7847, -1.0265, 1.6, -0.4, 1.57, 0.0], a=1.7, v=2.0, r=0.08)
  movej([0.7832, -1.0353, 1.6, -0.4, 1.57, 0.0], a=1.7, v=2.0, r=0.08)
  movej([0.7817, -1.0441, 1.6, -0.4, 1.57, 0.0], a=1.7, v=2.0, r=0.08)
  movej([0.7803, -1.053, 1.6, -0.4, 1.57, 0.0], a=1.7, v=2.0, r=0.08)
  movej([0.7789, -1.0619, 1.6, -0.4, 1.57, 0.0], a=1.7, v=2.0, r=0.08)
  movej([0.7775, -1.071, 1.6, -0.4, 1.57, 0.0], a=1.7, v=2.0, r=0.08)
  movej([0.7762, -1.0801, 1.6, -0.4, 1.57, 0.0], a=1.7, v=2.0, r=0.08)
  movej([0.775, -1.0892, 1.6, -0.4, 1.57, 0.0], a=1.7, v=2.0, r=0.08)
  movej([0.7738, -1.0984, 1.6, -0.4, 1.57, 0.0], a=1.7, v=2.0, r=0.08)
  movej([0.7726, -1.1077, 1.6, -0.4, 1.57, 0.0], a=1.7, v=2.0, r=0.08)
  movej([0.7715, -1.117, 1.6, -0.4, 1.57, 0.0], a=1.7, v=2.0, r=0.08)
  movej([0.7705, -1.1264, 1.6, -0.4, 1.57, 0.0], a=1.7, v=2.0, r=0.08)
  movej([0.7695, -1.1358, 1.6, -0.4, 1.57, 0.0], a=1.7, v=2.0, r=0.08)
  movej([0.7686, -1.1453, 1.6, -0.4, 1.57, 0.0], a=1.7, v=2.0, r=0.08)
  movej([0.7677, -1.1548, 1.6, -0.4, 1.57, 0.0], a=1.7, v=2.0, r=0.08)
  movej([0.7668, -1.1643, 1.6, -0.4, 1.57, 0.0], a=1.7, v=2.0, r=0.08)
  movej([0.766, -1.1739, 1.6, -0.4, 1.57, 0.0], a=1.7, v=2.0, r=0.08)
  movej([0.7653, -1.1836, 1.6, -0.4, 1.57, 0.0], a=1.7, v=2.0, r=0.08)
  movej([0.7646, -1.1932, 1.6, -0.4, 1.57, 0.0], a=1.7, v=2.0, r=0.08)
  movej([0.7639, -1.2029, 1.6, -0.4, 1.57, 0.0], a=1.7, v=2.0, r=0.08)
  movej([0.7633, -1.2127, 1.6, -0.4, 1.57, 0.0], a=1.7, v=2.0, r=0.08)
  movej([0.7628, -1.2224, 1.6, -0.4, 1.57, 0.0], a=1.7, v=2.0, r=0.08)
  movej([0.7623, -1.2322, 1.6, -0.4, 1.57, 0.0], a=1.7, v=2.0, r=0.08)
  movej([0.7618, -1.242, 1.6, -0.4, 1.57, 0.0], a=1.7, v=2.0, r=0.08)
  movej([0.7614, -1.2519, 1.6, -0.4, 1.57, 0.0], a=1.7, v=2.0, r=0.08)
  movej([0.7611, -1.2617, 1.6, -0.4, 1.57, 0.0], a=1.7, v=2.0, r=0.08)
  movej([0.7608, -1.2716, 1.6, -0.4, 1.57, 0.0], a=1.7, v=2.0, r=0.08)
  movej([0.7605, -1.2814, 1.6, -0.4, 1.57, 0.0], a=1.7, v=2.0, r=0.08)
  movej([0.7603, -1.2913, 1.6, -0.4, 1.57, 0.0], a=1.7, v=2.0, r=0.08)
  movej([0.7602, -1.3012, 1.6, -0.4, 1.57, 0.0], a=1.7, v=2.0, r=0.08)
  movej([0.7601, -1.3111, 1.6, -0.4, 1.57, 0.0], a=1.7, v=2.0, r=0.08)
  movej([0.76, -1.321, 1.6, -0.4, 1.57, 0.0], a=1.7, v=2.0, r=0.08)
  movej([0.76, -1.331, 1.6, -0.4, 1.57, 0.0], a=1.7, v=2.0, r=0.08)
  movej([0.7601, -1.3409, 1.6, -0.4, 1.57, 0.0], a=1.7, v=2.0, r=0.08)
  movej([0.7602, -1.3508, 1.6, -0.4, 1.57, 0.0], a=1.7, v=2.0, r=0.08)
  movej([0.7603, -1.3607, 1.6, -0.4, 1.57, 0.0], a=1.7, v=2.0, r=0.08)
  movej([0.7605, -1.3706, 1.6, -0.4, 1.57, 0.0], a=1.7, v=2.0, r=0.08)
  movej([0.7608, -1.3804, 1.6, -0.4, 1.57, 0.0], a=1.7, v=2.0, r=0.08)
  movej([0.7611, -1.3903, 1.6, -0.4, 1.57, 0.0], a=1.7, v=2.0, r=0.08)
  movej([0.7614, -1.4001, 1.6, -0.4, 1.57, 0.0], a=1.7, v=2.0, r=0.08)
  movej([0.7618, -1.41, 1.6, -0.4, 1.57, 0.0], a=1.7, v=2.0, r=0.08)
  movej([0.7623, -1.4198, 1.6, -0.4, 1.57, 0.0], a=1.7, v=2.0, r=0.08)
  movej([0.7628, -1.4296, 1.6, -0.4, 1.57, 0.0], a=1.7, v=2.0, r=0.08)
  movej([0.7633, -1.4393, 1.6, -0.4, 1.57, 0.0], a=1.7, v=2.0, r=0.08)
  movej([0.7639, -1.4491, 1.6, -0.4, 1.57, 0.0], a=1.7, v=2.0, r=0.08)
  movej([0.7646, -1.4588, 1.6, -0.4, 1.57, 0.0], a=1.7, v=2.0, r=0.08)
  movej([0.7653, -1.4684, 1.6, -0.4, 1.57, 0.0], a=1.7, v=2.0, r=0.08)
  movej([0.766, -1.4781, 1.6, -0.4, 1.57, 0.0], a=1.7, v=2.0, r=0.08)
  movej([0.7668, -1.4877, 1.6, -0.4, 1.57, 0.0], a=1.7, v=2.0, r=0.08)
  movej([0.7677, -1.4972, 1.6, -0.4, 1.57, 0.0], a=1.7, v=2.0, r=0.08)
  movej([0.7686, -1.5067, 1.6, -0.4, 1.57, 0.0], a=1.7, v=2.0, r=0.08)
  movej([0.7695, -1.5162, 1.6, -0.4, 1.57, 0.0], a=1.7, v=2.0, r=0.08)
  movej([0.7705, -1.5256, 1.6, -0.4, 1.57, 0.0], a=1.7, v=2.0, r=0.08)
  movej([0.7715, -1.535, 1.6, -0.4, 1.57, 0.0], a=1.7, v=2.0, r=0.08)
  movej([0.7726, -1.5443, 1.6, -0.4, 1.57, 0.0], a=1.7, v=2.0, r=0.08)
  movej([0.7738, -1.5536, 1.6, -0.4, 1.57, 0.0], a=1.7, v=2.0, r=0.08)
  movej([0.775, -1.5628, 1.6, -0.4, 1.57, 0.0], a=1.7, v=2.0, r=0.08)
  movej([0.7762, -1.5719, 1.6, -0.4, 1.57, 0.0], a=1.7, v=2.0, r=0.08)
  movej([0.7775, -1.581, 1.6, -0.4, 1.57, 0.0], a=1.7, v=2.0, r=0.08)
  movej([0.7789, -1.5901, 1.6, -0.4, 1.57, 0.0], a=1.7, v=2.0, r=0.08)
  movej([0.7803, -1.599, 1.6, -0.4, 1.57, 0.0], a=1.7, v=2.0, r=0.08)
  movej([0.7817, -1.6079, 1.6, -0.4, 1.57, 0.0], a=1.7, v=2.0, r=0.08)
  movej([0.7832, -1.6167, 1.6, -0.4, 1.57, 0.0], a=1.7, v=2.0, r=0.08)
  movej([0.7847, -1.6255, 1.6, -0.4, 1.57, 0.0], a=1.7, v=2.0, r=0.08)
  movej([0.7863, -1.6342, 1.6, -0.4, 1.57, 0.0], a=1.7, v=2.0, r=0.08)
  movej([0.7879, -1.6428, 1.6, -0.4, 1.57, 0.0], a=1.7, v=2.0, r=0.08)
  movej([0.7896, -1.6513, 1.6, -0.4, 1.57, 0.0], a=1.7, v=2.0, r=0.08)
  movej([0.7914, -1.6598, 1.6, -0.4, 1.57, 0.0], a=1.7, v=2.0, r=0.08)
  movej([0.7931, -1.6681, 1.6, -0.4, 1.57, 0.0], a=1.7, v=2.0, r=0.08)
  movej([0.795, -1.6764, 1.6, -0.4, 1.57, 0.0], a=1.7, v=2.0, r=0.08)
  movej([0.7968, -1.6846, 1.6, -0.4, 1.57, 0.0], a=1.7, v=2.0, r=0.08)
  movej([0.7988, -1.6927, 1.6, -0.4, 1.57, 0.0], a=1.7, v=2.0, r=0.08)
  movej([0.8007, -1.7007, 1.6, -0.4, 1.57, 0.0], a=1.7, v=2.0, r=0.08)
  movej([0.8027, -1.7086, 1.6, -0.4, 1.57, 0.0], a=1.7, v=2.0, r=0.08)
  movej([0.8048, -1.7164, 1.6, -0.4, 1.57, 0.0], a=1.7, v=2.0, r=0.08)
  movej([0.8069, -1.7242, 1.6, -0.4, 1.57, 0.0], a=1.7, v=2.0, r=0.08)
  movej([0.8091, -1.7318, 1.6, -0.4, 1.57, 0.0], a=1.7, v=2.0, r=0.08)
  movej([0.8113, -1.7393, 1.6, -0.4, 1.57, 0.0], a=1.7, v=2.0, r=0.08)
  movej([0.8135, -1.7468, 1.6, -0.4, 1.57, 0.0], a=1.7, v=2.0, r=0.08)
  movej([0.8158, -1.7541, 1.6, -0.4, 1.57, 0.0], a=1.7, v=2.0, r=0.08)
  movej([0.8182, -1.7613, 1.6, -0.4, 1.57, 0.0], a=1.7, v=2.0, r=0.08)
  movej([0.8206, -1.7684, 1.6, -0.4, 1.57, 0.0], a=1.7, v=2.0, r=0.08)
  movej([0.823, -1.7754, 1.6, -0.4, 1.57, 0.0], a=1.7, v=2.0, r=0.08)
  movej([0.8255, -1.7823, 1.6, -0.4, 1.57, 0.0], a=1.7, v=2.0, r=0.08)
  movej([0.828, -1.7891, 1.6, -0.4, 1.57, 0.0], a=1.7, v=2.0, r=0.08)
  movej([0.8306, -1.7957, 1.6, -0.4, 1.57, 0.0], a=1.7, v=2.0, r=0.08)
  movej([0.8333, -1.8023, 1.6, -0.4, 1.57, 0.0], a=1.7, v=2.0, r=0.08)
  movej([0.8359, -1.8087, 1.6, -0.4, 1.57, 0.0], a=1.7, v=2.0, r=0.08)
  movej([0.8386, -1.815, 1.6, -0.4, 1.57, 0.0], a=1.7, v=2.0, r=0.08)
  movej([0.8414, -1.8212, 1.6, -0.4, 1.57, 0.0], a=1.7, v=2.0, r=0.08)
  movej([0.8442, -1.8273, 1.6, -0.4, 1.57, 0.0], a=1.7, v=2.0, r=0.08)
  movej([0.8471, -1.8332, 1.6, -0.4, 1.57, 0.0], a=1.7, v=2.0, r=0.08)
  movej([0.8499, -1.839, 1.6, -0.4, 1.57, 0.0], a=1.7, v=2.0, r=0.08)
  movej([0.8529, -1.8447, 1.6, -0.4, 1.57, 0.0], a=1.7, v=2.0, r=0.08)
  movej([0.8559, -1.8503, 1.6, -0.4, 1.57, 0.0], a=1.7, v=2.0, r=0.08)
  movej([0.8589, -1.8557, 1.6, -0.4, 1.57, 0.0], a=1.7, v=2.0, r=0.08)
  movej([0.862, -1.861, 1.6, -0.4, 1.57, 0.0], a=1.7, v=2.0, r=0.08)
  movej([0.8651, -1.8662, 1.6, -0.4, 1.57, 0.0], a=1.7, v=2.0, r=0.08)
  movej([0.8682, -1.8712, 1.6, -0.4, 1.57, 0.0], a=1.7, v=2.0, r=0.08)
  movej([0.8715, -1.8761, 1.6, -0.4, 1.57, 0.0], a=1.7, v=2.0, r=0.08)
  movej([0.8747, -1.8808, 1.6, -0.4, 1.57, 0.0], a=1.7, v=2.0, r=0.08)
  movej([0.878, -1.8855, 1.6, -0.4, 1.57, 0.0], a=1.7, v=2.0, r=0.08)
  movej([0.8813, -1.89, 1.6, -0.4, 1.57, 0.0], a=1.7, v=2.0, r=0.08)
  movej([0.8847, -1.8943, 1.6, -0.4, 1.57, 0.0], a=1.7, v=2.0, r=0.08)
  movej([0.8881, -1.8985, 1.6, -0.4, 1.57, 0.0], a=1.7, v=2.0, r=0.08)
  movej([0.8916, -1.9026, 1.6, -0.4, 1.57, 0.0], a=1.7, v=2.0, r=0.08)
  movej([0.8951, -1.9065, 1.6, -0.4, 1.57, 0.0], a=1.7, v=2.0, r=0.08)
  movej([0.8986, -1.9103, 1.6, -0.4, 1.57, 0.0], a=1.7, v=2.0, r=0.08)
  movej([0.9022, -1.9139, 1.6, -0.4, 1.57, 0.0], a=1.7, v=2.0, r=0.08)
  movej([0.9058, -1.9174, 1.6, -0.4, 1.57, 0.0], a=1.7, v=2.0, r=0.08)
  movej([0.9095, -1.9207, 1.6, -0.4, 1.57, 0.0], a=1.7, v=2.0, r=0.08)
  movej([0.9132, -1.9239, 1.6, -0.4, 1.57, 0.0], a=1.7, v=2.0, r=0.08)
  movej([0.9169, -1.927, 1.6, -0.4, 1.57, 0.0], a=1.7, v=2.0, r=0.08)
  movej([0.9207, -1.9299, 1.6, -0.4, 1.57, 0.0], a=1.7, v=2.0, r=0.08)
  movej([0.9246, -1.9326, 1.6, -0.4, 1.57, 0.0], a=1.7, v=2.0, r=0.08)
  movej([0.9284, -1.9352, 1.6, -0.4, 1.57, 0.0], a=1.7, v=2.0, r=0.08)
  movej([0.9323, -1.9377, 1.6, -0.4, 1.57, 0.0], a=1.7, v=2.0, r=0.08)
  movej([0.9363, -1.94, 1.6, -0.4, 1.57, 0.0], a=1.7, v=2.0, r=0.08)
  movej([0.9403, -1.9421, 1.6, -0.4, 1.57, 0.0], a=1.7, v=2.0, r=0.08)
  movej([0.9443, -1.9441, 1.6, -0.4, 1.57, 0.0], a=1.7, v=2.0, r=0.08)
  movej([0.9484, -1.9459, 1.6, -0.4, 1.57, 0.0], a=1.7, v=2.0, r=0.08)
  movej([0.9525, -1.9476, 1.6, -0.4, 1.57, 0.0], a=1.7, v=2.0, r=0.08)
  movej([0.9566, -1.9492, 1.6, -0.4, 1.57, 0.0], a=1.7, v=2.0, r=0.08)
  movej([0.9608, -1.9505, 1.6, -0.4, 1.57, 0.0], a=1.7, v=2.0, r=0.08)
  movej([0.965, -1.9518, 1.6, -0.4, 1.57, 0.0], a=1.7, v=2.0, r=0.08)
  movej([0.9693, -1.9528, 1.6, -0.4, 1.57, 0.0], a=1.7, v=2.0, r=0.08)
  movej([0.9735, -1.9538, 1.6, -0.4, 1.57, 0.0], a=1.7, v=2.0, r=0.08)
  movej([0.9779, -1.9545, 1.6, -0.4, 1.57, 0.0], a=1.7, v=2.0, r=0.08)
  movej([0.9822, -1.9551, 1.6, -0.4, 1.57, 0.0], a=1.7, v=2.0, r=0.08)
  movej([0.9866, -1.9556, 1.6, -0.4, 1.57, 0.0], a=1.7, v=2.0, r=0.08)
  movej([0.9911, -1.9559, 1.6, -0.4, 1.57, 0.0], a=1.7, v=2.0, r=0.08)
  movej([0.9956, -1.956, 1.6, -0.4, 1.57, 0.0], a=1.7, v=2.0, r=0.08)
  movej([1.0001, -1.956, 1.6, -0.4, 1.57, 0.0], a=1.7, v=2.0, r=0.08)
  movej([1.0046, -1.9558, 1.6, -0.4, 1.57, 0.0], a=1.7, v=2.0, r=0.08)
  movej([1.0092, -1.9555, 1.6, -0.4, 1.57, 0.0], a=1.7, v=2.0, r=0.08)
  movej([1.0138, -1.955, 1.6, -0.4, 1.57, 0.0], a=1.7, v=2.0, r=0.08)
  movej([1.0184, -1.9543, 1.6, -0.4, 1.57, 0.0], a=1.7, v=2.0, r=0.08)
  movej([1.0231, -1.9535, 1.6, -0.4, 1.57, 0.0], a=1.7, v=2.0, r=0.08)
  movej([1.0278, -1.9526, 1.6, -0.4, 1.57, 0.0], a=1.7, v=2.0, r=0.08)
  movej([1.0326, -1.9515, 1.6, -0.4, 1.57, 0.0], a=1.7, v=2.0, r=0.08)
  movej([1.0374, -1.9502, 1.6, -0.4, 1.57, 0.0], a=1.7, v=2.0, r=0.08)
  movej([1.0422, -1.9488, 1.6, -0.4, 1.57, 0.0], a=1.7, v=2.0, r=0.08)
  movej([1.047, -1.9472, 1.6, -0.4, 1.57, 0.0], a=1.7, v=2.0, r=0.08)
  movej([1.0519, -1.9455, 1.6, -0.4, 1.57, 0.0], a=1.7, v=2.0, r=0.08)
  movej([1.0568, -1.9436, 1.6, -0.4, 1.57, 0.0], a=1.7, v=2.0, r=0.08)
  movej([1.0618, -1.9416, 1.6, -0.4, 1.57, 0.0], a=1.7, v=2.0, r=0.08)
  movej([1.0667, -1.9394, 1.6, -0.4, 1.57, 0.0], a=1.7, v=2.0, r=0.08)
  movej([1.0718, -1.9371, 1.6, -0.4, 1.57, 0.0], a=1.7, v=2.0, r=0.08)
  movej([1.0768, -1.9346, 1.6, -0.4, 1.57, 0.0], a=1.7, v=2.0, r=0.08)
  movej([1.0819, -1.932, 1.6, -0.4, 1.57, 0.0], a=1.7, v=2.0, r=0.08)
  movej([1.087, -1.9292, 1.6, -0.4, 1.57, 0.0], a=1.7, v=2.0, r=0.08)
  movej([1.0921, -1.9262, 1.6, -0.4, 1.57, 0.0], a=1.7, v=2.0, r=0.08)
  movej([1.0972, -1.9231, 1.6, -0.4, 1.57, 0.0], a=1.7, v=2.0, r=0.08)
  movej([1.1024, -1.9199, 1.6, -0.4, 1.57, 0.0], a=1.7, v=2.0, r=0.08)
  movej([1.1076, -1.9165, 1.6, -0.4, 1.57, 0.0], a=1.7, v=2.0, r=0.08)
  movej([1.1129, -1.913, 1.6, -0.4, 1.57, 0.0], a=1.7, v=2.0, r=0.08)
  movej([1.1182, -1.9093, 1.6, -0.4, 1.57, 0.0], a=1.7, v=2.0, r=0.08)
  movej([1.1235, -1.9055, 1.6, -0.4, 1.57, 0.0], a=1.7, v=2.0, r=0.08)
  movej([1.1288, -1.9016, 1.6, -0.4, 1.57, 0.0], a=1.7, v=2.0, r=0.08)
  movej([1.1341, -1.8975, 1.6, -0.4, 1.57, 0.0], a=1.7, v=2.0, r=0.08)
  movej([1.1395, -1.8932, 1.6, -0.4, 1.57, 0.0], a=1.7, v=2.0, r=0.08)
  movej([1.1449, -1.8888, 1.6, -0.4, 1.57, 0.0], a=1.7, v=2.0, r=0.08)
  movej([1.1504, -1.8843, 1.6, -0.4, 1.57, 0.0], a=1.7, v=2.0, r=0.08)
  movej([1.1558, -1.8797, 1.6, -0.4, 1.57, 0.0], a=1.7, v=2.0, r=0.08)
  movej([1.1613, -1.8749, 1.6, -0.4, 1.57, 0.0], a=1.7, v=2.0, r=0.08)
  movej([1.1668, -1.8699, 1.6, -0.4, 1.57, 0.0], a=1.7, v=2.0, r=0.08)
  movej([1.1724, -1.8649, 1.6, -0.4, 1.57, 0.0], a=1.7, v=2.0, r=0.08)
  movej([1.1779, -1.8597, 1.6, -0.4, 1.57, 0.0], a=1.7, v=2.0, r=0.08)
  movej([1.1835, -1.8543, 1.6, -0.4, 1.57, 0.0], a=1.7, v=2.0, r=0.08)
  movej([1.1891, -1.8489, 1.6, -0.4, 1.57, 0.0], a=1.7, v=2.0, r=0.08)
  movej([1.1948, -1.8433, 1.6, -0.4, 1.57, 0.0], a=1.7, v=2.0, r=0.08)
  movej([1.2004, -1.8376, 1.6, -0.4, 1.57, 0.0], a=1.7, v=2.0, r=0.08)
  movej([1.2061, -1.8317, 1.6, -0.4, 1.57, 0.0], a=1.7, v=2.0, r=0.08)
  movej([1.2118, -1.8258, 1.6, -0.4, 1.57, 0.0], a=1.7, v=2.0, r=0.08)
  movej([1.2175, -1.8197, 1.6, -0.4, 1.57, 0.0], a=1.7, v=2.0, r=0.08)
  movej([1.2233, -1.8134, 1.6, -0.4, 1.57, 0.0], a=1.7, v=2.0, r=0.08)
  movej([1.229, -1.8071, 1.6, -0.4, 1.57, 0.0], a=1.7, v=2.0, r=0.08)
  movej([1.2348, -1.8006, 1.6, -0.4, 1.57, 0.0], a=1.7, v=2.0, r=0.08)
  movej([1.2406, -1.7941, 1.6, -0.4, 1.57, 0.0], a=1.7, v=2.0, r=0.08)
  movej([1.2465, -1.7874, 1.6, -0.4, 1.57, 0.0], a=1.7, v=2.0, r=0.08)
  movej([1.2523, -1.7806, 1.6, -0.4, 1.57, 0.0], a=1.7, v=2.0, r=0.08)
  movej([1.2582, -1.7737, 1.6, -0.4, 1.57, 0.0], a=1.7, v=2.0, r=0.08)
  movej([1.2641, -1.7666, 1.6, -0.4, 1.57, 0.0], a=1.7, v=2.0, r=0.08)
  movej([1.27, -1.7595, 1.6, -0.4, 1.57, 0.0], a=1.7, v=2.0, r=0.08)
  movej([1.2759, -1.7523, 1.6, -0.4, 1.57, 0.0], a=1.7, v=2.0, r=0.08)
  movej([1.2818, -1.7449, 1.6, -0.4, 1.57, 0.0], a=1.7, v=2.0, r=0.08)
  movej([1.2878, -1.7375, 1.6, -0.4, 1.57, 0.0], a=1.7, v=2.0, r=0.08)
  movej([1.2938, -1.7299, 1.6, -0.4, 1.57, 0.0], a=1.7, v=2.0, r=0.08)
  movej([1.2998, -1.7222, 1.6, -0.4, 1.57, 0.0], a=1.7, v=2.0, r=0.08)
  movej([1.3058, -1.7145, 1.6, -0.4, 1.57, 0.0], a=1.7, v=2.0, r=0.08)
  movej([1.3118, -1.7066, 1.6, -0.4, 1.57, 0.0], a=1.7, v=2.0, r=0.08)
  movej([1.3179, -1.6987, 1.6, -0.4, 1.57, 0.0], a=1.7, v=2.0, r=0.08)
  movej([1.3239, -1.6907, 1.6, -0.4, 1.57, 0.0], a=1.7, v=2.0, r=0.08)
  movej([1.33, -1.6825, 1.6, -0.4, 1.57, 0.0], a=1.7, v=2.0, r=0.08)
  movej([1.3361, -1.6743, 1.6, -0.4, 1.57, 0.0], a=1.7, v=2.0, r=0.08)
  movej([1.3422, -1.666, 1.6, -0.4, 1.57, 0.0], a=1.7, v=2.0, r=0.08)
  movej([1.3483, -1.6577, 1.6, -0.4, 1.57, 0.0], a=1.7, v=2.0, r=0.08)
  movej([1.3545, -1.6492, 1.6, -0.4, 1.57, 0.0], a=1.7, v=2.0, r=0.08)
  movej([1.3606, -1.6406, 1.6, -0.4, 1.57, 0.0], a=1.7, v=2.0, r=0.08)
  movej([1.3668, -1.632, 1.6, -0.4, 1.57, 0.0], a=1.7, v=2.0, r=0.08)
  movej([1.3729, -1.6233, 1.6, -0.4, 1.57, 0.0], a=1.7, v=2.0, r=0.08)
  movej([1.3791, -1.6145, 1.6, -0.4, 1.57, 0.0], a=1.7, v=2.0, r=0.08)
  movej([1.3853, -1.6057, 1.6, -0.4, 1.57, 0.0], a=1.7, v=2.0, r=0.08)
  movej([1.3915, -1.5968, 1.6, -0.4, 1.57, 0.0], a=1.7, v=2.0, r=0.08)
  movej([1.3977, -1.5878, 1.6, -0.4, 1.57, 0.0], a=1.7, v=2.0, r=0.08)
  movej([1.404, -1.5788, 1.6, -0.4, 1.57, 0.0], a=1.7, v=2.0, r=0.08)
  movej([1.4102, -1.5697, 1.6, -0.4, 1.57, 0.0], a=1.7, v=2.0, r=0.08)
  movej([1.4165, -1.5605, 1.6, -0.4, 1.57, 0.0], a=1.7, v=2.0, r=0.08)
  movej([1.4227, -1.5513, 1.6, -0.4, 1.57, 0.0], a=1.7, v=2.0, r=0.08)
  movej([1.429, -1.542, 1.6, -0.4, 1.57, 0.0], a=1.7, v=2.0, r=0.08)
  movej([1.4353, -1.5327, 1.6, -0.4, 1.57, 0.0], a=1.7, v=2.0, r=0.08)
  movej([1.4416, -1.5233, 1.6, -0.4, 1.57, 0.0], a=1.7, v=2.0, r=0.08)
  movej([1.4478, -1.5138, 1.6, -0.4, 1.57, 0.0], a=1.7, v=2.0, r=0.08)
  movej([1.4541, -1.5044, 1.6, -0.4, 1.57, 0.0], a=1.7, v=2.0, r=0.08)
  movej([1.4605, -1.4948, 1.6, -0.4, 1.57, 0.0], a=1.7, v=2.0, r=0.08)
  movej([1.4668, -1.4853, 1.6, -0.4, 1.57, 0.0], a=1.7, v=2.0, r=0.08)
  movej([1.4731, -1.4757, 1.6, -0.4, 1.57, 0.0], a=1.7, v=2.0, r=0.08)
  movej([1.4794, -1.466, 1.6, -0.4, 1.57, 0.0], a=1.7, v=2.0, r=0.08)
  movej([1.4858, -1.4563, 1.6, -0.4, 1.57, 0.0], a=1.7, v=2.0, r=0.08)
  movej([1.4921, -1.4466, 1.6, -0.4, 1.57, 0.0], a=1.7, v=2.0, r=0.08)
  movej([1.4984, -1.4369, 1.6, -0.4, 1.57, 0.0], a=1.7, v=2.0, r=0.08)
  movej([1.5048, -1.4271, 1.6, -0.4, 1.57, 0.0], a=1.7, v=2.0, r=0.08)
  movej([1.5111, -1.4173, 1.6, -0.4, 1.57, 0.0], a=1.7, v=2.0, r=0.08)
  movej([1.5175, -1.4075, 1.6, -0.4, 1.57, 0.0], a=1.7, v=2.0, r=0.08)
  movej([1.5238, -1.3977, 1.6, -0.4, 1.57, 0.0], a=1.7, v=2.0, r=0.08)
  movej([1.5302, -1.3878, 1.6, -0.4, 1.57, 0.0], a=1.7, v=2.0, r=0.08)
  movej([1.5366, -1.378, 1.6, -0.4, 1.57, 0.0], a=1.7, v=2.0, r=0.08)
  movej([1.5429, -1.3681, 1.6, -0.4, 1.57, 0.0], a=1.7, v=2.0, r=0.08)
  movej([1.5493, -1.3582, 1.6, -0.4, 1.57, 0.0], a=1.7, v=2.0, r=0.08)
  movej([1.5557, -1.3483, 1.6, -0.4, 1.57, 0.0], a=1.7, v=2.0, r=0.08)
  movej([1.562, -1.3384, 1.6, -0.4, 1.57, 0.0], a=1.7, v=2.0, r=0.08)
  movej([1.5684, -1.3285, 1.6, -0.4, 1.57, 0.0], a=1.7, v=2.0, r=0.08)
  movej([1.5748, -1.3186, 1.6, -0.4, 1.57, 0.0], a=1.7, v=2.0, r=0.08)
  movej([1.5811, -1.3087, 1.6, -0.4, 1.57, 0.0], a=1.7, v=2.0, r=0.08)
  movej([1.5875, -1.2988, 1.6, -0.4, 1.57, 0.0], a=1.7, v=2.0, r=0.08)
  movej([1.5939, -1.2889, 1.6, -0.4, 1.57, 0.0], a=1.7, v=2.0, r=0.08)
  movej([1.6002, -1.279, 1.6, -0.4, 1.57, 0.0], a=1.7, v=2.0, r=0.08)
  movej([1.6066, -1.2691, 1.6, -0.4, 1.57, 0.0], a=1.7, v=2.0, r=0.08)
  movej([1.613, -1.2592, 1.6, -0.4, 1.57, 0.0], a=1.7, v=2.0, r=0.08)
  movej([1.6193, -1.2494, 1.6, -0.4, 1.57, 0.0], a=1.7, v=2.0, r=0.08)
  movej([1.6257, -1.2396, 1.6, -0.4, 1.57, 0.0], a=1.7, v=2.0, r=0.08)
  movej([1.632, -1.2298, 1.6, -0.4, 1.57, 0.0], a=1.7, v=2.0, r=0.08)
  movej([1.6384, -1.22, 1.6, -0.4, 1.57, 0.0], a=1.7, v=2.0, r=0.08)
  movej([1.6447, -1.2102, 1.6, -0.4, 1.57, 0.0], a=1.7, v=2.0, r=0.08)
  movej([1.6511, -1.2005, 1.6, -0.4, 1.57, 0.0], a=1.7, v=2.0, r=0.08)
  movej([1.6574, -1.1908, 1.6, -0.4, 1.57, 0.0], a=1.7, v=2.0, r=0.08)
  movej([1.6637, -1.1812, 1.6, -0.4, 1.57, 0.0], a=1.7, v=2.0, r=0.08)
  movej([1.6701, -1.1715, 1.6, -0.4, 1.57, 0.0], a=1.7, v=2.0, r=0.08)
  movej([1.6764, -1.1619, 1.6, -0.4, 1.57, 0.0], a=1.7, v=2.0, r=0.08)
  movej([1.6827, -1.1524, 1.6, -0.4, 1.57, 0.0], a=1.7, v=2.0, r=0.08)
  movej([1.689, -1.1429, 1.6, -0.4, 1.57, 0.0], a=1.7, v=2.0, r=0.08)
  movej([1.6953, -1.1334, 1.6, -0.4, 1.57, 0.0], a=1.7, v=2.0, r=0.08)
  movej([1.7016, -1.124, 1.6, -0.4, 1.57, 0.0], a=1.7, v=2.0, r=0.08)
  movej([1.7079, -1.1147, 1.6, -0.4, 1.57, 0.0], a=1.7, v=2.0, r=0.08)
  movej([1.7141, -1.1054, 1.6, -0.4, 1.57, 0.0], a=1.7, v=2.0, r=0.08)
  movej([1.7204, -1.0961, 1.6, -0.4, 1.57, 0.0], a=1.7, v=2.0, r=0.08)
  movej([1.7267, -1.0869, 1.6, -0.4, 1.57, 0.0], a=1.7, v=2.0, r=0.08)
  movej([1.7329, -1.0778, 1.6, -0.4, 1.57, 0.0], a=1.7, v=2.0, r=0.08)
  movej([1.7391, -1.0687, 1.6, -0.4, 1.57, 0.0], a=1.7, v=2.0, r=0.08)
  movej([1.7454, -1.0597, 1.6, -0.4, 1.57, 0.0], a=1.7, v=2.0, r=0.08)
  movej([1.7516, -1.0507, 1.6, -0.4, 1.57, 0.0], a=1.7, v=2.0, r=0.08)
  movej([1.7578, -1.0419, 1.6, -0.4, 1.57, 0.0], a=1.7, v=2.0, r=0.08)
  movej([1.764, -1.0331, 1.6, -0.4, 1.57, 0.0], a=1.7, v=2.0, r=0.08)
  movej([1.7701, -1.0243, 1.6, -0.4, 1.57, 0.0], a=1.7, v=2.0, r=0.08)
  movej([1.7763, -1.0157, 1.6, -0.4, 1.57, 0.0], a=1.7, v=2.0, r=0.08)
  movej([1.7825, -1.0071, 1.6, -0.4, 1.57, 0.0], a=1.7, v=2.0, r=0.08)
  movej([1.7886, -0.9986, 1.6, -0.4, 1.57, 0.0], a=1.7, v=2.0, r=0.08)
  movej([1.7947, -0.9901, 1.6, -0.4, 1.57, 0.0], a=1.7, v=2.0, r=0.08)
  movej([1.8008, -0.9818, 1.6, -0.4, 1.57, 0.0], a=1.7, v=2.0, r=0.08)
  movej([1.8069, -0.9735, 1.6, -0.4, 1.57, 0.0], a=1.7, v=2.0, r=0.08)
  movej([1.813, -0.9654, 1.6, -0.4, 1.57, 0.0], a=1.7, v=2.0, r=0.08)
  movej([1.8191, -0.9573, 1.6, -0.4, 1.57, 0.0], a=1.7, v=2.0, r=0.08)
  movej([1.8251, -0.9493, 1.6, -0.4, 1.57, 0.0], a=1.7, v=2.0, r=0.08)
  movej([1.8312, -0.9414, 1.6, -0.4, 1.57, 0.0], a=1.7, v=2.0, r=0.08)
  movej([1.8372, -0.9336, 1.6, -0.4, 1.57, 0.0], a=1.7, v=2.0, r=0.08)
  movej([1.8432, -0.9259, 1.6, -0.4, 1.57, 0.0], a=1.7, v=2.0, r=0.08)
  movej([1.8492, -0.9183, 1.6, -0.4, 1.57, 0.0], a=1.7, v=2.0, r=0.08)
  movej([1.8552, -0.9108, 1.6, -0.4, 1.57, 0.0], a=1.7, v=2.0, r=0.08)
  movej([1.8611, -0.9034, 1.6, -0.4, 1.57, 0.0], a=1.7, v=2.0, r=0.08)
  movej([1.8671, -0.8961, 1.6, -0.4, 1.57, 0.0], a=1.7, v=2.0, r=0.08)
  movej([1.873, -0.8889, 1.6, -0.4, 1.57, 0.0], a=1.7, v=2.0, r=0.08)
  movej([1.8789, -0.8818, 1.6, -0.4, 1.57, 0.0], a=1.7, v=2.0, r=0.08)
  movej([1.8847, -0.8749, 1.6, -0.4, 1.57, 0.0], a=1.7, v=2.0, r=0.08)
  movej([1.8906, -0.868, 1.6, -0.4, 1.57, 0.0], a=1.7, v=2.0, r=0.08)
  movej([1.8964, -0.8613, 1.6, -0.4, 1.57, 0.0], a=1.7, v=2.0, r=0.08)
  movej([1.9023, -0.8546, 1.6, -0.4, 1.57, 0.0], a=1.7, v=2.0, r=0.08)
  movej([1.9081, -0.8481, 1.6, -0.4, 1.57, 0.0], a=1.7, v=2.0, r=0.08)
  movej([1.9138, -0.8417, 1.6, -0.4, 1.57, 0.0], a=1.7, v=2.0, r=0.08)
  movej([1.9196, -0.8354, 1.6, -0.4, 1.57, 0.0], a=1.7, v=2.0, r=0.08)
  movej([1.9253, -0.8293, 1.6, -0.4, 1.57, 0.0], a=1.7, v=2.0, r=0.08)
  movej([1.931, -0.8232, 1.6, -0.4, 1.57, 0.0], a=1.7, v=2.0, r=0.08)
  movej([1.9367, -0.8173, 1.6, -0.4, 1.57, 0.0], a=1.7, v=2.0, r=0.08)
  movej([1.9424, -0.8116, 1.6, -0.4, 1.57, 0.0], a=1.7, v=2.0, r=0.08)
  movej([1.9481, -0.8059, 1.6, -0.4, 1.57, 0.0], a=1.7, v=2.0, r=0.08)
  movej([1.9537, -0.8004, 1.6, -0.4, 1.57, 0.0], a=1.7, v=2.0, r=0.08)
  movej([1.9593, -0.795, 1.6, -0.4, 1.57, 0.0], a=1.7, v=2.0, r=0.08)
  movej([1.9648, -0.7897, 1.6, -0.4, 1.57, 0.0], a=1.7, v=2.0, r=0.08)
  movej([1.9704, -0.7846, 1.6, -0.4, 1.57, 0.0], a=1.7, v=2.0, r=0.08)
  movej([1.9759, -0.7796, 1.6, -0.4, 1.57, 0.0], a=1.7, v=2.0, r=0.08)
  movej([1.9814, -0.7747, 1.6, -0.4, 1.57, 0.0], a=1.7, v=2.0, r=0.08)
  movej([1.9869, -0.77, 1.6, -0.4, 1.57, 0.0], a=1.7, v=2.0, r=0.08)
  movej([1.9923, -0.7654, 1.6, -0.4, 1.57, 0.0], a=1.7, v=2.0, r=0.08)
  movej([1.9978, -0.7609, 1.6, -0.4, 1.57, 0.0], a=1.7, v=2.0, r=0.08)
  movej([2.0032, -0.7566, 1.6, -0.4, 1.57, 0.0], a=1.7, v=2.0, r=0.08)
  movej([2.0085, -0.7525, 1.6, -0.4, 1.57, 0.0], a=1.7, v=2.0, r=0.08)
  movej([2.0139, -0.7484, 1.6, -0.4, 1.57, 0.0], a=1.7, v=2.0, r=0.08)
  movej([2.0192, -0.7445, 1.6, -0.4, 1.57, 0.0], a=1.7, v=2.0, r=0.08)
  movej([2.0245, -0.7408, 1.6, -0.4, 1.57, 0.0], a=1.7, v=2.0, r=0.08)
  movej([2.0297, -0.7372, 1.6, -0.4, 1.57, 0.0], a=1.7, v=2.0, r=0.08)
  movej([2.035, -0.7338, 1.6, -0.4, 1.57, 0.0], a=1.7, v=2.0, r=0.08)
  movej([2.0402, -0.7305, 1.6, -0.4, 1.57, 0.0], a=1.7, v=2.0, r=0.08)
  movej([2.0453, -0.7273, 1.6, -0.4, 1.57, 0.0], a=1.7, v=2.0, r=0.08)
  movej([2.0505, -0.7243, 1.6, -0.4, 1.57, 0.0], a=1.7, v=2.0, r=0.08)
  movej([2.0556, -0.7214, 1.6, -0.4, 1.57, 0.0], a=1.7, v=2.0, r=0.08)
  movej([2.0607, -0.7187, 1.6, -0.4, 1.57, 0.0], a=1.7, v=2.0, r=0.08)
  movej([2.0657, -0.7162, 1.6, -0.4, 1.57, 0.0], a=1.7, v=2.0, r=0.08)
  movej([2.0707, -0.7137, 1.6, -0.4, 1.57, 0.0], a=1.7, v=2.0, r=0.08)
  movej([2.0757, -0.7115, 1.6, -0.4, 1.57, 0.0], a=1.7, v=2.0, r=0.08)
  movej([2.0807, -0.7094, 1.6, -0.4, 1.57, 0.0], a=1.7, v=2.0, r=0.08)
  movej([2.0856, -0.7074, 1.6, -0.4, 1.57, 0.0], a=1.7, v=2.0, r=0.08)
  movej([2.0905, -0.7056, 1.6, -0.4, 1.57, 0.0], a=1.7, v=2.0, r=0.08)
  movej([2.0954, -0.704, 1.6, -0.4, 1.57, 0.0], a=1.7, v=2.0, r=0.08)
  movej([2.1002, -0.7025, 1.6, -0.4, 1.57, 0.0], a=1.7, v=2.0, r=0.08)
  movej([2.105, -0.7011, 1.6, -0.4, 1.57, 0.0], a=1.7, v=2.0, r=0.08)
  movej([2.1098, -0.7, 1.6, -0.4, 1.57, 0.0], a=1.7, v=2.0, r=0.08)
  movej([2.1145, -0.6989, 1.6, -0.4, 1.57, 0.0], a=1.7, v=2.0, r=0.08)
  movej([2.1192, -0.698, 1.6, -0.4, 1.57, 0.0], a=1.7, v=2.0, r=0.08)
  movej([2.1239, -0.6973, 1.6, -0.4, 1.57, 0.0], a=1.7, v=2.0, r=0.08)
  movej([2.1285, -0.6968, 1.6, -0.4, 1.57, 0.0], a=1.7, v=2.0, r=0.08)
  movej([2.1331, -0.6964, 1.6, -0.4, 1.57, 0.0], a=1.7, v=2.0, r=0.08)
  movej([2.1377, -0.6961, 1.6, -0.4, 1.57, 0.0], a=1.7, v=2.0, r=0.08)
  movej([2.1422, -0.696, 1.6, -0.4, 1.57, 0.0], a=1.7, v=2.0, r=0.08)
  movej([2.1467, -0.6961, 1.6, -0.4, 1.57, 0.0], a=1.7, v=2.0, r=0.08)
  movej([2.1511, -0.6963, 1.6, -0.4, 1.57, 0.0], a=1.7, v=2.0, r=0.08)
  movej([2.1556, -0.6966, 1.6, -0.4, 1.57, 0.0], a=1.7, v=2.0, r=0.08)
  movej([2.1599, -0.6972, 1.6, -0.4, 1.57, 0.0], a=1.7, v=2.0, r=0.08)
  movej([2.1643, -0.6978, 1.6, -0.4, 1.57, 0.0], a=1.7, v=2.0, r=0.08)
  movej([2.1686, -0.6987, 1.6, -0.4, 1.57, 0.0], a=1.7, v=2.0, r=0.08)
  movej([2.1729, -0.6997, 1.6, -0.4, 1.57, 0.0], a=1.7, v=2.0, r=0.08)
  movej([2.1771, -0.7008, 1.6, -0.4, 1.57, 0.0], a=1.7, v=2.0, r=0.08)
  movej([2.1813, -0.7021, 1.6, -0.4, 1.57, 0.0], a=1.7, v=2.0, r=0.08)
  movej([2.1855, -0.7036, 1.6, -0.4, 1.57, 0.0], a=1.7, v=2.0, r=0.08)
  movej([2.1896, -0.7052, 1.6, -0.4, 1.57, 0.0], a=1.7, v=2.0, r=0.08)
  movej([2.1937, -0.707, 1.6, -0.4, 1.57, 0.0], a=1.7, v=2.0, r=0.08)
  movej([2.1977, -0.7089, 1.6, -0.4, 1.57, 0.0], a=1.7, v=2.0, r=0.08)
  movej([2.2017, -0.7109, 1.6, -0.4, 1.57, 0.0], a=1.7, v=2.0, r=0.08)
  movej([2.2057, -0.7132, 1.6, -0.4, 1.57, 0.0], a=1.7, v=2.0, r=0.08)
  movej([2.2096, -0.7155, 1.6, -0.4, 1.57, 0.0], a=1.7, v=2.0, r=0.08)
  movej([2.2135, -0.7181, 1.6, -0.4, 1.57, 0.0], a=1.7, v=2.0, r=0.08)
  movej([2.2174, -0.7207, 1.6, -0.4, 1.57, 0.0], a=1.7, v=2.0, r=0.08)
  movej([2.2212, -0.7236, 1.6, -0.4, 1.57, 0.0], a=1.7, v=2.0, r=0.08)
  movej([2.2249, -0.7265, 1.6, -0.4, 1.57, 0.0], a=1.7, v=2.0, r=0.08)
  movej([2.2287, -0.7296, 1.6, -0.4, 1.57, 0.0], a=1.7, v=2.0, r=0.08)
  movej([2.2323, -0.7329, 1.6, -0.4, 1.57, 0.0], a=1.7, v=2.0, r=0.08)
  movej([2.236, -0.7363, 1.6, -0.4, 1.57, 0.0], a=1.7, v=2.0, r=0.08)
  movej([2.2396, -0.7399, 1.6, -0.4, 1.57, 0.0], a=1.7, v=2.0, r=0.08)
  movej([2.2432, -0.7436, 1.6, -0.4, 1.57, 0.0], a=1.7, v=2.0, r=0.08)
  movej([2.2467, -0.7475, 1.6, -0.4, 1.57, 0.0], a=1.7, v=2.0, r=0.08)
  movej([2.2502, -0.7514, 1.6, -0.4, 1.57, 0.0], a=1.7, v=2.0, r=0.08)
  movej([2.2536, -0.7556, 1.6, -0.4, 1.57, 0.0], a=1.7, v=2.0, r=0.08)
  movej([2.257, -0.7599, 1.6, -0.4, 1.57, 0.0], a=1.7, v=2.0, r=0.08)
  movej([2.2603, -0.7643, 1.6, -0.4, 1.57, 0.0], a=1.7, v=2.0, r=0.08)
  movej([2.2637, -0.7688, 1.6, -0.4, 1.57, 0.0], a=1.7, v=2.0, r=0.08)
  movej([2.2669, -0.7735, 1.6, -0.4, 1.57, 0.0], a=1.7, v=2.0, r=0.08)
  movej([2.2701, -0.7784, 1.6, -0.4, 1.57, 0.0], a=1.7, v=2.0, r=0.08)
  movej([2.2733, -0.7833, 1.6, -0.4, 1.57, 0.0], a=1.7, v=2.0, r=0.08)
  movej([2.2765, -0.7884, 1.6, -0.4, 1.57, 0.0], a=1.7, v=2.0, r=0.08)
  movej([2.2796, -0.7936, 1.6, -0.4, 1.57, 0.0], a=1.7, v=2.0, r=0.08)
  movej([2.2826, -0.799, 1.6, -0.4, 1.57, 0.0], a=1.7, v=2.0, r=0.08)
  movej([2.2856, -0.8045, 1.6, -0.4, 1.57, 0.0], a=1.7, v=2.0, r=0.08)
  movej([2.2886, -0.8101, 1.6, -0.4, 1.57, 0.0], a=1.7, v=2.0, r=0.08)
  movej([2.2915, -0.8159, 1.6, -0.4, 1.57, 0.0], a=1.7, v=2.0, r=0.08)
  movej([2.2944, -0.8218, 1.6, -0.4, 1.57, 0.0], a=1.7, v=2.0, r=0.08)
  movej([2.2972, -0.8278, 1.6, -0.4, 1.57, 0.0], a=1.7, v=2.0, r=0.08)
  movej([2.3, -0.8339, 1.6, -0.4, 1.57, 0.0], a=1.7, v=2.0, r=0.08)
  movej([2.3027, -0.8401, 1.6, -0.4, 1.57, 0.0], a=1.7, v=2.0, r=0.08)
  movej([2.3054, -0.8465, 1.6, -0.4, 1.57, 0.0], a=1.7, v=2.0, r=0.08)
  movej([2.3081, -0.853, 1.6, -0.4, 1.57, 0.0], a=1.7, v=2.0, r=0.08)
  movej([2.3107, -0.8596, 1.6, -0.4, 1.57, 0.0], a=1.7, v=2.0, r=0.08)
  movej([2.3132, -0.8663, 1.6, -0.4, 1.57, 0.0], a=1.7, v=2.0, r=0.08)
  movej([2.3157, -0.8731, 1.6, -0.4, 1.57, 0.0], a=1.7, v=2.0, r=0.08)
  movej([2.3182, -0.8801, 1.6, -0.4, 1.57, 0.0], a=1.7, v=2.0, r=0.08)
  movej([2.3206, -0.8871, 1.6, -0.4, 1.57, 0.0], a=1.7, v=2.0, r=0.08)
  movej([2.323, -0.8943, 1.6, -0.4, 1.57, 0.0], a=1.7, v=2.0, r=0.08)
  movej([2.3253, -0.9016, 1.6, -0.4, 1.57, 0.0], a=1.7, v=2.0, r=0.08)
  movej([2.3276, -0.9089, 1.6, -0.4, 1.57, 0.0], a=1.7, v=2.0, r=0.08)
  movej([2.3298, -0.9164, 1.6, -0.4, 1.57, 0.0], a=1.7, v=2.0, r=0.08)
  movej([2.332, -0.924, 1.6, -0.4, 1.57, 0.0], a=1.7, v=2.0, r=0.08)
  movej([2.3341, -0.9317, 1.6, -0.4, 1.57, 0.0], a=1.7, v=2.0, r=0.08)
  movej([2.3362, -0.9395, 1.6, -0.4, 1.57, 0.0], a=1.7, v=2.0, r=0.08)
  movej([2.3383, -0.9473, 1.6, -0.4, 1.57, 0.0], a=1.7, v=2.0, r=0.08)
  movej([2.3403, -0.9553, 1.6, -0.4, 1.57, 0.0], a=1.7, v=2.0, r=0.08)
  movej([2.3422, -0.9634, 1.6, -0.4, 1.57, 0.0], a=1.7, v=2.0, r=0.08)
  movej([2.3441, -0.9715, 1.6, -0.4, 1.57, 0.0], a=1.7, v=2.0, r=0.08)
  movej([2.346, -0.9797, 1.6, -0.4, 1.57, 0.0], a=1.7, v=2.0, r=0.08)
  movej([2.3478, -0.9881, 1.6, -0.4, 1.57, 0.0], a=1.7, v=2.0, r=0.08)
  movej([2.3495, -0.9965, 1.6, -0.4, 1.57, 0.0], a=1.7, v=2.0, r=0.08)
  movej([2.3512, -1.0049, 1.6, -0.4, 1.57, 0.0], a=1.7, v=2.0, r=0.08)
  movej([2.3529, -1.0135, 1.6, -0.4, 1.57, 0.0], a=1.7, v=2.0, r=0.08)
  movej([2.3545, -1.0221, 1.6, -0.4, 1.57, 0.0], a=1.7, v=2.0, r=0.08)
  movej([2.3561, -1.0309, 1.6, -0.4, 1.57, 0.0], a=1.7, v=2.0, r=0.08)
  movej([2.3576, -1.0397, 1.6, -0.4, 1.57, 0.0], a=1.7, v=2.0, r=0.08)
  movej([2.359, -1.0485, 1.6, -0.4, 1.57, 0.0], a=1.7, v=2.0, r=0.08)
  movej([2.3604, -1.0574, 1.6, -0.4, 1.57, 0.0], a=1.7, v=2.0, r=0.08)
  movej([2.3618, -1.0664, 1.6, -0.4, 1.57, 0.0], a=1.7, v=2.0, r=0.08)
  movej([2.3631, -1.0755, 1.6, -0.4, 1.57, 0.0], a=1.7, v=2.0, r=0.08)
  movej([2.3644, -1.0846, 1.6, -0.4, 1.57, 0.0], a=1.7, v=2.0, r=0.08)
  movej([2.3656, -1.0938, 1.6, -0.4, 1.57, 0.0], a=1.7, v=2.0, r=0.08)
  movej([2.3668, -1.103, 1.6, -0.4, 1.57, 0.0], a=1.7, v=2.0, r=0.08)
  movej([2.3679, -1.1123, 1.6, -0.4, 1.57, 0.0], a=1.7, v=2.0, r=0.08)
  movej([2.369, -1.1217, 1.6, -0.4, 1.57, 0.0], a=1.7, v=2.0, r=0.08)
  movej([2.37, -1.1311, 1.6, -0.4, 1.57, 0.0], a=1.7, v=2.0, r=0.08)
  movej([2.371, -1.1405, 1.6, -0.4, 1.57, 0.0], a=1.7, v=2.0, r=0.08)
  movej([2.3719, -1.15, 1.6, -0.4, 1.57, 0.0], a=1.7, v=2.0, r=0.08)
  movej([2.3728, -1.1596, 1.6, -0.4, 1.57, 0.0], a=1.7, v=2.0, r=0.08)
  movej([2.3736, -1.1691, 1.6, -0.4, 1.57, 0.0], a=1.7, v=2.0, r=0.08)
  movej([2.3744, -1.1787, 1.6, -0.4, 1.57, 0.0], a=1.7, v=2.0, r=0.08)
  movej([2.3751, -1.1884, 1.6, -0.4, 1.57, 0.0], a=1.7, v=2.0, r=0.08)
  movej([2.3758, -1.1981, 1.6, -0.4, 1.57, 0.0], a=1.7, v=2.0, r=0.08)
  movej([2.3764, -1.2078, 1.6, -0.4, 1.57, 0.0], a=1.7, v=2.0, r=0.08)
  movej([2.377, -1.2176, 1.6, -0.4, 1.57, 0.0], a=1.7, v=2.0, r=0.08)
  movej([2.3775, -1.2273, 1.6, -0.4, 1.57, 0.0], a=1.7, v=2.0, r=0.08)
  movej([2.378, -1.2371, 1.6, -0.4, 1.57, 0.0], a=1.7, v=2.0, r=0.08)
  movej([2.3784, -1.2469, 1.6, -0.4, 1.57, 0.0], a=1.7, v=2.0, r=0.08)
  movej([2.3788, -1.2568, 1.6, -0.4, 1.57, 0.0], a=1.7, v=2.0, r=0.08)
  movej([2.3791, -1.2666, 1.6, -0.4, 1.57, 0.0], a=1.7, v=2.0, r=0.08)
  movej([2.3794, -1.2765, 1.6, -0.4, 1.57, 0.0], a=1.7, v=2.0, r=0.08)
  movej([2.3796, -1.2864, 1.6, -0.4, 1.57, 0.0], a=1.7, v=2.0, r=0.08)
  movej([2.3798, -1.2963, 1.6, -0.4, 1.57, 0.0], a=1.7, v=2.0, r=0.08)
  movej([2.3799, -1.3062, 1.6, -0.4, 1.57, 0.0], a=1.7, v=2.0, r=0.08)
  movej([2.38, -1.3161, 1.6, -0.4, 1.57, 0.0], a=1.7, v=2.0, r=0.08)
  movej([2.38, -1.326, 1.6, -0.4, 1.57, 0.0], a=1.7, v=2.0, r=0.08)
  movej([2.137, -1.326, 1.6, -0.4, 1.57, 0.0], a=1.7, v=2.0, r=0.08)
  movej([2.137, -1.3329, 1.6, -0.4, 1.57, 0.0], a=1.7, v=2.0, r=0.08)
  movej([2.1369, -1.3399, 1.6, -0.4, 1.57, 0.0], a=1.7, v=2.0, r=0.08)
  movej([2.1368, -1.3468, 1.6, -0.4, 1.57, 0.0], a=1.7, v=2.0, r=0.08)
  movej([2.1367, -1.3537, 1.6, -0.4, 1.57, 0.0], a=1.7, v=2.0, r=0.08)
  movej([2.1366, -1.3606, 1.6, -0.4, 1.57, 0.0], a=1.7, v=2.0, r=0.08)
  movej([2.1364, -1.3676, 1.6, -0.4, 1.57, 0.0], a=1.7, v=2.0, r=0.08)
  movej([2.1361, -1.3745, 1.6, -0.4, 1.57, 0.0], a=1.7, v=2.0, r=0.08)
  movej([2.1359, -1.3813, 1.6, -0.4, 1.57, 0.0], a=1.7, v=2.0, r=0.08)
  movej([2.1356, -1.3882, 1.6, -0.4, 1.57, 0.0], a=1.7, v=2.0, r=0.08)
  movej([2.1352, -1.3951, 1.6, -0.4, 1.57, 0.0], a=1.7, v=2.0, r=0.08)
  movej([2.1349, -1.4019, 1.6, -0.4, 1.57, 0.0], a=1.7, v=2.0, r=0.08)
  movej([2.1345, -1.4087, 1.6, -0.4, 1.57, 0.0], a=1.7, v=2.0, r=0.08)
  movej([2.134, -1.4155, 1.6, -0.4, 1.57, 0.0], a=1.7, v=2.0, r=0.08)
  movej([2.1336, -1.4223, 1.6, -0.4, 1.57, 0.0], a=1.7, v=2.0, r=0.08)
  movej([2.1331, -1.4291, 1.6, -0.4, 1.57, 0.0], a=1.7, v=2.0, r=0.08)
  movej([2.1325, -1.4358, 1.6, -0.4, 1.57, 0.0], a=1.7, v=2.0, r=0.08)
  movej([2.1319, -1.4425, 1.6, -0.4, 1.57, 0.0], a=1.7, v=2.0, r=0.08)
  movej([2.1313, -1.4492, 1.6, -0.4, 1.57, 0.0], a=1.7, v=2.0, r=0.08)
  movej([2.1307, -1.4558, 1.6, -0.4, 1.57, 0.0], a=1.7, v=2.0, r=0.08)
  movej([2.13, -1.4624, 1.6, -0.4, 1.57, 0.0], a=1.7, v=2.0, r=0.08)
  movej([2.1293, -1.469, 1.6, -0.4, 1.57, 0.0], a=1.7, v=2.0, r=0.08)
  movej([2.1285, -1.4756, 1.6, -0.4, 1.57, 0.0], a=1.7, v=2.0, r=0.08)
  movej([2.1278, -1.4821, 1.6, -0.4, 1.57, 0.0], a=1.7, v=2.0, r=0.08)
  movej([2.1269, -1.4885, 1.6, -0.4, 1.57, 0.0], a=1.7, v=2.0, r=0.08)
  movej([2.1261, -1.495, 1.6, -0.4, 1.57, 0.0], a=1.7, v=2.0, r=0.08)
  movej([2.1252, -1.5013, 1.6, -0.4, 1.57, 0.0], a=1.7, v=2.0, r=0.08)
  movej([2.1243, -1.5077, 1.6, -0.4, 1.57, 0.0], a=1.7, v=2.0, r=0.08)
  movej([2.1233, -1.514, 1.6, -0.4, 1.57, 0.0], a=1.7, v=2.0, r=0.08)
  movej([2.1223, -1.5202, 1.6, -0.4, 1.57, 0.0], a=1.7, v=2.0, r=0.08)
  movej([2.1213, -1.5264, 1.6, -0.4, 1.57, 0.0], a=1.7, v=2.0, r=0.08)
  movej([2.1202, -1.5326, 1.6, -0.4, 1.57, 0.0], a=1.7, v=2.0, r=0.08)
  movej([2.1191, -1.5387, 1.6, -0.4, 1.57, 0.0], a=1.7, v=2.0, r=0.08)
  movej([2.118, -1.5447, 1.6, -0.4, 1.57, 0.0], a=1.7, v=2.0, r=0.08)
  movej([2.1169, -1.5507, 1.6, -0.4, 1.57, 0.0], a=1.7, v=2.0, r=0.08)
  movej([2.1157, -1.5567, 1.6, -0.4, 1.57, 0.0], a=1.7, v=2.0, r=0.08)
  movej([2.1144, -1.5626, 1.6, -0.4, 1.57, 0.0], a=1.7, v=2.0, r=0.08)
  movej([2.1132, -1.5684, 1.6, -0.4, 1.57, 0.0], a=1.7, v=2.0, r=0.08)
  movej([2.1119, -1.5742, 1.6, -0.4, 1.57, 0.0], a=1.7, v=2.0, r=0.08)
  movej([2.1105, -1.5799, 1.6, -0.4, 1.57, 0.0], a=1.7, v=2.0, r=0.08)
  movej([2.1092, -1.5855, 1.6, -0.4, 1.57, 0.0], a=1.7, v=2.0, r=0.08)
  movej([2.1078, -1.5911, 1.6, -0.4, 1.57, 0.0], a=1.7, v=2.0, r=0.08)
  movej([2.1064, -1.5966, 1.6, -0.4, 1.57, 0.0], a=1.7, v=2.0, r=0.08)
  movej([2.1049, -1.602, 1.6, -0.4, 1.57, 0.0], a=1.7, v=2.0, r=0.08)
  movej([2.1034, -1.6074, 1.6, -0.4, 1.57, 0.0], a=1.7, v=2.0, r=0.08)
  movej([2.1019, -1.6127, 1.6, -0.4, 1.57, 0.0], a=1.7, v=2.0, r=0.08)
  movej([2.1003, -1.6179, 1.6, -0.4, 1.57, 0.0], a=1.7, v=2.0, r=0.08)
  movej([2.0987, -1.6231, 1.6, -0.4, 1.57, 0.0], a=1.7, v=2.0, r=0.08)
  movej([2.0971, -1.6282, 1.6, -0.4, 1.57, 0.0], a=1.7, v=2.0, r=0.08)
  movej([2.0954, -1.6332, 1.6, -0.4, 1.57, 0.0], a=1.7, v=2.0, r=0.08)
  movej([2.0937, -1.6381, 1.6, -0.4, 1.57, 0.0], a=1.7, v=2.0, r=0.08)
  movej([2.092, -1.643, 1.6, -0.4, 1.57, 0.0], a=1.7, v=2.0, r=0.08)
  movej([2.0903, -1.6478, 1.6, -0.4, 1.57, 0.0], a=1.7, v=2.0, r=0.08)
  movej([2.0885, -1.6525, 1.6, -0.4, 1.57, 0.0], a=1.7, v=2.0, r=0.08)
  movej([2.0866, -1.6571, 1.6, -0.4, 1.57, 0.0], a=1.7, v=2.0, r=0.08)
  movej([2.0848, -1.6616, 1.6, -0.4, 1.57, 0.0], a=1.7, v=2.0, r=0.08)
  movej([2.0829, -1.6661, 1.6, -0.4, 1.57, 0.0], a=1.7, v=2.0, r=0.08)
  movej([2.081, -1.6705, 1.6, -0.4, 1.57, 0.0], a=1.7, v=2.0, r=0.08)
  movej([2.079, -1.6748, 1.6, -0.4, 1.57, 0.0], a=1.7, v=2.0, r=0.08)
  movej([2.0771, -1.679, 1.6, -0.4, 1.57, 0.0], a=1.7, v=2.0, r=0.08)
  movej([2.075, -1.6831, 1.6, -0.4, 1.57, 0.0], a=1.7, v=2.0, r=0.08)
  movej([2.073, -1.6871, 1.6, -0.4, 1.57, 0.0], a=1.7, v=2.0, r=0.08)
  movej([2.0709, -1.691, 1.6, -0.4, 1.57, 0.0], a=1.7, v=2.0, r=0.08)
  movej([2.0688, -1.6949, 1.6, -0.4, 1.57, 0.0], a=1.7, v=2.0, r=0.08)
  movej([2.0667, -1.6986, 1.6, -0.4, 1.57, 0.0], a=1.7, v=2.0, r=0.08)
  movej([2.0645, -1.7023, 1.6, -0.4, 1.57, 0.0], a=1.7, v=2.0, r=0.08)
  movej([2.0623, -1.7059, 1.6, -0.4, 1.57, 0.0], a=1.7, v=2.0, r=0.08)
  movej([2.0601, -1.7094, 1.6, -0.4, 1.57, 0.0], a=1.7, v=2.0, r=0.08)
  movej([2.0578, -1.7127, 1.6, -0.4, 1.57, 0.0], a=1.7, v=2.0, r=0.08)
  movej([2.0556, -1.716, 1.6, -0.4, 1.57, 0.0], a=1.7, v=2.0, r=0.08)
  movej([2.0532, -1.7192, 1.6, -0.4, 1.57, 0.0], a=1.7, v=2.0, r=0.08)
  movej([2.0509, -1.7223, 1.6, -0.4, 1.57, 0.0], a=1.7, v=2.0, r=0.08)
  movej([2.0485, -1.7253, 1.6, -0.4, 1.57, 0.0], a=1.7, v=2.0, r=0.08)
  movej([2.0461, -1.7282, 1.6, -0.4, 1.57, 0.0], a=1.7, v=2.0, r=0.08)
  movej([2.0437, -1.731, 1.6, -0.4, 1.57, 0.0], a=1.7, v=2.0, r=0.08)
  movej([2.0412, -1.7337, 1.6, -0.4, 1.57, 0.0], a=1.7, v=2.0, r=0.08)
  movej([2.0387, -1.7363, 1.6, -0.4, 1.57, 0.0], a=1.7, v=2.0, r=0.08)
  movej([2.0362, -1.7388, 1.6, -0.4, 1.57, 0.0], a=1.7, v=2.0, r=0.08)
  movej([2.0336, -1.7412, 1.6, -0.4, 1.57, 0.0], a=1.7, v=2.0, r=0.08)
  movej([2.0311, -1.7434, 1.6, -0.4, 1.57, 0.0], a=1.7, v=2.0, r=0.08)
  movej([2.0284, -1.7456, 1.6, -0.4, 1.57, 0.0], a=1.7, v=2.0, r=0.08)
  movej([2.0258, -1.7477, 1.6, -0.4, 1.57, 0.0], a=1.7, v=2.0, r=0.08)
  movej([2.0231, -1.7497, 1.6, -0.4, 1.57, 0.0], a=1.7, v=2.0, r=0.08)
  movej([2.0205, -1.7516, 1.6, -0.4, 1.57, 0.0], a=1.7, v=2.0, r=0.08)
  movej([2.0177, -1.7533, 1.6, -0.4, 1.57, 0.0], a=1.7, v=2.0, r=0.08)
  movej([2.015, -1.755, 1.6, -0.4, 1.57, 0.0], a=1.7, v=2.0, r=0.08)
  movej([2.0122, -1.7565, 1.6, -0.4, 1.57, 0.0], a=1.7, v=2.0, r=0.08)
  movej([2.0094, -1.758, 1.6, -0.4, 1.57, 0.0], a=1.7, v=2.0, r=0.08)
  movej([2.0066, -1.7593, 1.6, -0.4, 1.57, 0.0], a=1.7, v=2.0, r=0.08)
  movej([2.0037, -1.7606, 1.6, -0.4, 1.57, 0.0], a=1.7, v=2.0, r=0.08)
  movej([2.0008, -1.7617, 1.6, -0.4, 1.57, 0.0], a=1.7, v=2.0, r=0.08)
  movej([1.9979, -1.7627, 1.6, -0.4, 1.57, 0.0], a=1.7, v=2.0, r=0.08)
  movej([1.995, -1.7636, 1.6, -0.4, 1.57, 0.0], a=1.7, v=2.0, r=0.08)
  movej([1.992, -1.7644, 1.6, -0.4, 1.57, 0.0], a=1.7, v=2.0, r=0.08)
  movej([1.989, -1.7651, 1.6, -0.4, 1.57, 0.0], a=1.7, v=2.0, r=0.08)
  movej([1.986, -1.7657, 1.6, -0.4, 1.57, 0.0], a=1.7, v=2.0, r=0.08)
  movej([1.983, -1.7662, 1.6, -0.4, 1.57, 0.0], a=1.7, v=2.0, r=0.08)
  movej([1.9799, -1.7666, 1.6, -0.4, 1.57, 0.0], a=1.7, v=2.0, r=0.08)
  movej([1.9768, -1.7668, 1.6, -0.4, 1.57, 0.0], a=1.7, v=2.0, r=0.08)
  movej([1.9737, -1.767, 1.6, -0.4, 1.57, 0.0], a=1.7, v=2.0, r=0.08)
  movej([1.9705, -1.767, 1.6, -0.4, 1.57, 0.0], a=1.7, v=2.0, r=0.08)
  movej([1.9674, -1.7669, 1.6, -0.4, 1.57, 0.0], a=1.7, v=2.0, r=0.08)
  movej([1.9642, -1.7668, 1.6, -0.4, 1.57, 0.0], a=1.7, v=2.0, r=0.08)
  movej([1.961, -1.7665, 1.6, -0.4, 1.57, 0.0], a=1.7, v=2.0, r=0.08)
  movej([1.9577, -1.7661, 1.6, -0.4, 1.57, 0.0], a=1.7, v=2.0, r=0.08)
  movej([1.9544, -1.7656, 1.6, -0.4, 1.57, 0.0], a=1.7, v=2.0, r=0.08)
  movej([1.9512, -1.765, 1.6, -0.4, 1.57, 0.0], a=1.7, v=2.0, r=0.08)
  movej([1.9478, -1.7642, 1.6, -0.4, 1.57, 0.0], a=1.7, v=2.0, r=0.08)
  movej([1.9445, -1.7634, 1.6, -0.4, 1.57, 0.0], a=1.7, v=2.0, r=0.08)
  movej([1.9412, -1.7625, 1.6, -0.4, 1.57, 0.0], a=1.7, v=2.0, r=0.08)
  movej([1.9378, -1.7614, 1.6, -0.4, 1.57, 0.0], a=1.7, v=2.0, r=0.08)
  movej([1.9344, -1.7603, 1.6, -0.4, 1.57, 0.0], a=1.7, v=2.0, r=0.08)
  movej([1.9309, -1.759, 1.6, -0.4, 1.57, 0.0], a=1.7, v=2.0, r=0.08)
  movej([1.9275, -1.7576, 1.6, -0.4, 1.57, 0.0], a=1.7, v=2.0, r=0.08)
  movej([1.924, -1.7562, 1.6, -0.4, 1.57, 0.0], a=1.7, v=2.0, r=0.08)
  movej([1.9205, -1.7546, 1.6, -0.4, 1.57, 0.0], a=1.7, v=2.0, r=0.08)
  movej([1.917, -1.7529, 1.6, -0.4, 1.57, 0.0], a=1.7, v=2.0, r=0.08)
  movej([1.9135, -1.7511, 1.6, -0.4, 1.57, 0.0], a=1.7, v=2.0, r=0.08)
  movej([1.9099, -1.7492, 1.6, -0.4, 1.57, 0.0], a=1.7, v=2.0, r=0.08)
  movej([1.9063, -1.7472, 1.6, -0.4, 1.57, 0.0], a=1.7, v=2.0, r=0.08)
  movej([1.9027, -1.7451, 1.6, -0.4, 1.57, 0.0], a=1.7, v=2.0, r=0.08)
  movej([1.8991, -1.7429, 1.6, -0.4, 1.57, 0.0], a=1.7, v=2.0, r=0.08)
  movej([1.8955, -1.7406, 1.6, -0.4, 1.57, 0.0], a=1.7, v=2.0, r=0.08)
  movej([1.8918, -1.7382, 1.6, -0.4, 1.57, 0.0], a=1.7, v=2.0, r=0.08)
  movej([1.8881, -1.7356, 1.6, -0.4, 1.57, 0.0], a=1.7, v=2.0, r=0.08)
  movej([1.8844, -1.733, 1.6, -0.4, 1.57, 0.0], a=1.7, v=2.0, r=0.08)
  movej([1.8807, -1.7303, 1.6, -0.4, 1.57, 0.0], a=1.7, v=2.0, r=0.08)
  movej([1.877, -1.7275, 1.6, -0.4, 1.57, 0.0], a=1.7, v=2.0, r=0.08)
  movej([1.8732, -1.7246, 1.6, -0.4, 1.57, 0.0], a=1.7, v=2.0, r=0.08)
  movej([1.8694, -1.7215, 1.6, -0.4, 1.57, 0.0], a=1.7, v=2.0, r=0.08)
  movej([1.8656, -1.7184, 1.6, -0.4, 1.57, 0.0], a=1.7, v=2.0, r=0.08)
  movej([1.8618, -1.7152, 1.6, -0.4, 1.57, 0.0], a=1.7, v=2.0, r=0.08)
  movej([1.858, -1.7119, 1.6, -0.4, 1.57, 0.0], a=1.7, v=2.0, r=0.08)
  movej([1.8541, -1.7085, 1.6, -0.4, 1.57, 0.0], a=1.7, v=2.0, r=0.08)
  movej([1.8503, -1.705, 1.6, -0.4, 1.57, 0.0], a=1.7, v=2.0, r=0.08)
  movej([1.8464, -1.7014, 1.6, -0.4, 1.57, 0.0], a=1.7, v=2.0, r=0.08)
  movej([1.8425, -1.6977, 1.6, -0.4, 1.57, 0.0], a=1.7, v=2.0, r=0.08)
  movej([1.8386, -1.6939, 1.6, -0.4, 1.57, 0.0], a=1.7, v=2.0, r=0.08)
  movej([1.8346, -1.6901, 1.6, -0.4, 1.57, 0.0], a=1.7, v=2.0, r=0.08)
  movej([1.8307, -1.6861, 1.6, -0.4, 1.57, 0.0], a=1.7, v=2.0, r=0.08)
  movej([1.8267, -1.6821, 1.6, -0.4, 1.57, 0.0], a=1.7, v=2.0, r=0.08)
  movej([1.8227, -1.6779, 1.6, -0.4, 1.57, 0.0], a=1.7, v=2.0, r=0.08)
  movej([1.8187, -1.6737, 1.6, -0.4, 1.57, 0.0], a=1.7, v=2.0, r=0.08)
  movej([1.8147, -1.6694, 1.6, -0.4, 1.57, 0.0], a=1.7, v=2.0, r=0.08)
  movej([1.8107, -1.665, 1.6, -0.4, 1.57, 0.0], a=1.7, v=2.0, r=0.08)
  movej([1.8066, -1.6605, 1.6, -0.4, 1.57, 0.0], a=1.7, v=2.0, r=0.08)
  movej([1.8026, -1.656, 1.6, -0.4, 1.57, 0.0], a=1.7, v=2.0, r=0.08)
  movej([1.7985, -1.6513, 1.6, -0.4, 1.57, 0.0], a=1.7, v=2.0, r=0.08)
  movej([1.7944, -1.6466, 1.6, -0.4, 1.57, 0.0], a=1.7, v=2.0, r=0.08)
  movej([1.7903, -1.6418, 1.6, -0.4, 1.57, 0.0], a=1.7, v=2.0, r=0.08)
  movej([1.7862, -1.6369, 1.6, -0.4, 1.57, 0.0], a=1.7, v=2.0, r=0.08)
  movej([1.7821, -1.632, 1.6, -0.4, 1.57, 0.0], a=1.7, v=2.0, r=0.08)
  movej([1.7779, -1.6269, 1.6, -0.4, 1.57, 0.0], a=1.7, v=2.0, r=0.08)
  movej([1.7738, -1.6218, 1.6, -0.4, 1.57, 0.0], a=1.7, v=2.0, r=0.08)
  movej([1.7696, -1.6166, 1.6, -0.4, 1.57, 0.0], a=1.7, v=2.0, r=0.08)
  movej([1.7654, -1.6114, 1.6, -0.4, 1.57, 0.0], a=1.7, v=2.0, r=0.08)
  movej([1.7612, -1.6061, 1.6, -0.4, 1.57, 0.0], a=1.7, v=2.0, r=0.08)
  movej([1.757, -1.6007, 1.6, -0.4, 1.57, 0.0], a=1.7, v=2.0, r=0.08)
  movej([1.7528, -1.5952, 1.6, -0.4, 1.57, 0.0], a=1.7, v=2.0, r=0.08)
  movej([1.7486, -1.5897, 1.6, -0.4, 1.57, 0.0], a=1.7, v=2.0, r=0.08)
  movej([1.7444, -1.5841, 1.6, -0.4, 1.57, 0.0], a=1.7, v=2.0, r=0.08)
  movej([1.7401, -1.5784, 1.6, -0.4, 1.57, 0.0], a=1.7, v=2.0, r=0.08)
  movej([1.7359, -1.5727, 1.6, -0.4, 1.57, 0.0], a=1.7, v=2.0, r=0.08)
  movej([1.7316, -1.5669, 1.6, -0.4, 1.57, 0.0], a=1.7, v=2.0, r=0.08)
  movej([1.7273, -1.5611, 1.6, -0.4, 1.57, 0.0], a=1.7, v=2.0, r=0.08)
  movej([1.723, -1.5552, 1.6, -0.4, 1.57, 0.0], a=1.7, v=2.0, r=0.08)
  movej([1.7187, -1.5492, 1.6, -0.4, 1.57, 0.0], a=1.7, v=2.0, r=0.08)
  movej([1.7144, -1.5432, 1.6, -0.4, 1.57, 0.0], a=1.7, v=2.0, r=0.08)
  movej([1.7101, -1.5372, 1.6, -0.4, 1.57, 0.0], a=1.7, v=2.0, r=0.08)
  movej([1.7058, -1.5311, 1.6, -0.4, 1.57, 0.0], a=1.7, v=2.0, r=0.08)
  movej([1.7014, -1.5249, 1.6, -0.4, 1.57, 0.0], a=1.7, v=2.0, r=0.08)
  movej([1.6971, -1.5187, 1.6, -0.4, 1.57, 0.0], a=1.7, v=2.0, r=0.08)
  movej([1.6927, -1.5124, 1.6, -0.4, 1.57, 0.0], a=1.7, v=2.0, r=0.08)
  movej([1.6884, -1.5061, 1.6, -0.4, 1.57, 0.0], a=1.7, v=2.0, r=0.08)
  movej([1.684, -1.4998, 1.6, -0.4, 1.57, 0.0], a=1.7, v=2.0, r=0.08)
  movej([1.6797, -1.4934, 1.6, -0.4, 1.57, 0.0], a=1.7, v=2.0, r=0.08)
  movej([1.6753, -1.4869, 1.6, -0.4, 1.57, 0.0], a=1.7, v=2.0, r=0.08)
  movej([1.6709, -1.4804, 1.6, -0.4, 1.57, 0.0], a=1.7, v=2.0, r=0.08)
  movej([1.6665, -1.4739, 1.6, -0.4, 1.57, 0.0], a=1.7, v=2.0, r=0.08)
  movej([1.6621, -1.4674, 1.6, -0.4, 1.57, 0.0], a=1.7, v=2.0, r=0.08)
  movej([1.6577, -1.4608, 1.6, -0.4, 1.57, 0.0], a=1.7, v=2.0, r=0.08)
  movej([1.6533, -1.4542, 1.6, -0.4, 1.57, 0.0], a=1.7, v=2.0, r=0.08)
  movej([1.6489, -1.4475, 1.6, -0.4, 1.57, 0.0], a=1.7, v=2.0, r=0.08)
  movej([1.6445, -1.4408, 1.6, -0.4, 1.57, 0.0], a=1.7, v=2.0, r=0.08)
  movej([1.64, -1.4341, 1.6, -0.4, 1.57, 0.0], a=1.7, v=2.0, r=0.08)
  movej([1.6356, -1.4274, 1.6, -0.4, 1.57, 0.0], a=1.7, v=2.0, r=0.08)
  movej([1.6312, -1.4206, 1.6, -0.4, 1.57, 0.0], a=1.7, v=2.0, r=0.08)
  movej([1.6268, -1.4138, 1.6, -0.4, 1.57, 0.0], a=1.7, v=2.0, r=0.08)
  movej([1.6223, -1.407, 1.6, -0.4, 1.57, 0.0], a=1.7, v=2.0, r=0.08)
  movej([1.6179, -1.4002, 1.6, -0.4, 1.57, 0.0], a=1.7, v=2.0, r=0.08)
  movej([1.6134, -1.3934, 1.6, -0.4, 1.57, 0.0], a=1.7, v=2.0, r=0.08)
  movej([1.609, -1.3865, 1.6, -0.4, 1.57, 0.0], a=1.7, v=2.0, r=0.08)
  movej([1.6045, -1.3796, 1.6, -0.4, 1.57, 0.0], a=1.7, v=2.0, r=0.08)
  movej([1.6001, -1.3727, 1.6, -0.4, 1.57, 0.0], a=1.7, v=2.0, r=0.08)
  movej([1.5956, -1.3658, 1.6, -0.4, 1.57, 0.0], a=1.7, v=2.0, r=0.08)
  movej([1.5912, -1.3589, 1.6, -0.4, 1.57, 0.0], a=1.7, v=2.0, r=0.08)
  movej([1.5867, -1.352, 1.6, -0.4, 1.57, 0.0], a=1.7, v=2.0, r=0.08)
  movej([1.5823, -1.3451, 1.6, -0.4, 1.57, 0.0], a=1.7, v=2.0, r=0.08)
  movej([1.5778, -1.3381, 1.6, -0.4, 1.57, 0.0], a=1.7, v=2.0, r=0.08)
  movej([1.5733, -1.3312, 1.6, -0.4, 1.57, 0.0], a=1.7, v=2.0, r=0.08)
  movej([1.5689, -1.3243, 1.6, -0.4, 1.57, 0.0], a=1.7, v=2.0, r=0.08)
  movej([1.5644, -1.3173, 1.6, -0.4, 1.57, 0.0], a=1.7, v=2.0, r=0.08)
  movej([1.56, -1.3104, 1.6, -0.4, 1.57, 0.0], a=1.7, v=2.0, r=0.08)
  movej([1.5555, -1.3035, 1.6, -0.4, 1.57, 0.0], a=1.7, v=2.0, r=0.08)
  movej([1.5511, -1.2965, 1.6, -0.4, 1.57, 0.0], a=1.7, v=2.0, r=0.08)
  movej([1.5466, -1.2896, 1.6, -0.4, 1.57, 0.0], a=1.7, v=2.0, r=0.08)
  movej([1.5421, -1.2827, 1.6, -0.4, 1.57, 0.0], a=1.7, v=2.0, r=0.08)
  movej([1.5377, -1.2758, 1.6, -0.4, 1.57, 0.0], a=1.7, v=2.0, r=0.08)
  movej([1.5332, -1.2689, 1.6, -0.4, 1.57, 0.0], a=1.7, v=2.0, r=0.08)
  movej([1.5288, -1.2621, 1.6, -0.4, 1.57, 0.0], a=1.7, v=2.0, r=0.08)
  movej([1.5243, -1.2552, 1.6, -0.4, 1.57, 0.0], a=1.7, v=2.0, r=0.08)
  movej([1.5199, -1.2484, 1.6, -0.4, 1.57, 0.0], a=1.7, v=2.0, r=0.08)
  movej([1.5155, -1.2416, 1.6, -0.4, 1.57, 0.0], a=1.7, v=2.0, r=0.08)
  movej([1.511, -1.2348, 1.6, -0.4, 1.57, 0.0], a=1.7, v=2.0, r=0.08)
  movej([1.5066, -1.228, 1.6, -0.4, 1.57, 0.0], a=1.7, v=2.0, r=0.08)
  movej([1.5022, -1.2212, 1.6, -0.4, 1.57, 0.0], a=1.7, v=2.0, r=0.08)
  movej([1.4977, -1.2145, 1.6, -0.4, 1.57, 0.0], a=1.7, v=2.0, r=0.08)
  movej([1.4933, -1.2078, 1.6, -0.4, 1.57, 0.0], a=1.7, v=2.0, r=0.08)
  movej([1.4889, -1.2012, 1.6, -0.4, 1.57, 0.0], a=1.7, v=2.0, r=0.08)
  movej([1.4845, -1.1945, 1.6, -0.4, 1.57, 0.0], a=1.7, v=2.0, r=0.08)
  movej([1.4801, -1.1879, 1.6, -0.4, 1.57, 0.0], a=1.7, v=2.0, r=0.08)
  movej([1.4757, -1.1813, 1.6, -0.4, 1.57, 0.0], a=1.7, v=2.0, r=0.08)
  movej([1.4713, -1.1748, 1.6, -0.4, 1.57, 0.0], a=1.7, v=2.0, r=0.08)
  movej([1.4669, -1.1683, 1.6, -0.4, 1.57, 0.0], a=1.7, v=2.0, r=0.08)
  movej([1.4625, -1.1619, 1.6, -0.4, 1.57, 0.0], a=1.7, v=2.0, r=0.08)
  movej([1.4582, -1.1554, 1.6, -0.4, 1.57, 0.0], a=1.7, v=2.0, r=0.08)
  movej([1.4538, -1.1491, 1.6, -0.4, 1.57, 0.0], a=1.7, v=2.0, r=0.08)
  movej([1.4494, -1.1427, 1.6, -0.4, 1.57, 0.0], a=1.7, v=2.0, r=0.08)
  movej([1.4451, -1.1364, 1.6, -0.4, 1.57, 0.0], a=1.7, v=2.0, r=0.08)
  movej([1.4407, -1.1302, 1.6, -0.4, 1.57, 0.0], a=1.7, v=2.0, r=0.08)
  movej([1.4364, -1.124, 1.6, -0.4, 1.57, 0.0], a=1.7, v=2.0, r=0.08)
  movej([1.4321, -1.1179, 1.6, -0.4, 1.57, 0.0], a=1.7, v=2.0, r=0.08)
  movej([1.4277, -1.1118, 1.6, -0.4, 1.57, 0.0], a=1.7, v=2.0, r=0.08)
  movej([1.4234, -1.1057, 1.6, -0.4, 1.57, 0.0], a=1.7, v=2.0, r=0.08)
  movej([1.4191, -1.0998, 1.6, -0.4, 1.57, 0.0], a=1.7, v=2.0, r=0.08)
  movej([1.4148, -1.0938, 1.6, -0.4, 1.57, 0.0], a=1.7, v=2.0, r=0.08)
  movej([1.4105, -1.088, 1.6, -0.4, 1.57, 0.0], a=1.7, v=2.0, r=0.08)
  movej([1.4063, -1.0822, 1.6, -0.4, 1.57, 0.0], a=1.7, v=2.0, r=0.08)
  movej([1.402, -1.0764, 1.6, -0.4, 1.57, 0.0], a=1.7, v=2.0, r=0.08)
  movej([1.3978, -1.0707, 1.6, -0.4, 1.57, 0.0], a=1.7, v=2.0, r=0.08)
  movej([1.3935, -1.0651, 1.6, -0.4, 1.57, 0.0], a=1.7, v=2.0, r=0.08)
  movej([1.3893, -1.0595, 1.6, -0.4, 1.57, 0.0], a=1.7, v=2.0, r=0.08)
  movej([1.3851, -1.0541, 1.6, -0.4, 1.57, 0.0], a=1.7, v=2.0, r=0.08)
  movej([1.3809, -1.0486, 1.6, -0.4, 1.57, 0.0], a=1.7, v=2.0, r=0.08)
  movej([1.3767, -1.0433, 1.6, -0.4, 1.57, 0.0], a=1.7, v=2.0, r=0.08)
  movej([1.3725, -1.038, 1.6, -0.4, 1.57, 0.0], a=1.7, v=2.0, r=0.08)
  movej([1.3683, -1.0328, 1.6, -0.4, 1.57, 0.0], a=1.7, v=2.0, r=0.08)
  movej([1.3641, -1.0276, 1.6, -0.4, 1.57, 0.0], a=1.7, v=2.0, r=0.08)
  movej([1.36, -1.0226, 1.6, -0.4, 1.57, 0.0], a=1.7, v=2.0, r=0.08)
  movej([1.3558, -1.0176, 1.6, -0.4, 1.57, 0.0], a=1.7, v=2.0, r=0.08)
  movej([1.3517, -1.0126, 1.6, -0.4, 1.57, 0.0], a=1.7, v=2.0, r=0.08)
  movej([1.3476, -1.0078, 1.6, -0.4, 1.57, 0.0], a=1.7, v=2.0, r=0.08)
  movej([1.3435, -1.003, 1.6, -0.4, 1.57, 0.0], a=1.7, v=2.0, r=0.08)
  movej([1.3394, -0.9983, 1.6, -0.4, 1.57, 0.0], a=1.7, v=2.0, r=0.08)
  movej([1.3354, -0.9937, 1.6, -0.4, 1.57, 0.0], a=1.7, v=2.0, r=0.08)
  movej([1.3313, -0.9892, 1.6, -0.4, 1.57, 0.0], a=1.7, v=2.0, r=0.08)
  movej([1.3273, -0.9848, 1.6, -0.4, 1.57, 0.0], a=1.7, v=2.0, r=0.08)
  movej([1.3233, -0.9804, 1.6, -0.4, 1.57, 0.0], a=1.7, v=2.0, r=0.08)
  movej([1.3193, -0.9762, 1.6, -0.4, 1.57, 0.0], a=1.7, v=2.0, r=0.08)
  movej([1.3153, -0.972, 1.6, -0.4, 1.57, 0.0], a=1.7, v=2.0, r=0.08)
  movej([1.3113, -0.9679, 1.6, -0.4, 1.57, 0.0], a=1.7, v=2.0, r=0.08)
  movej([1.3073, -0.9639, 1.6, -0.4, 1.57, 0.0], a=1.7, v=2.0, r=0.08)
  movej([1.3034, -0.96, 1.6, -0.4, 1.57, 0.0], a=1.7, v=2.0, r=0.08)
  movej([1.2995, -0.9562, 1.6, -0.4, 1.57, 0.0], a=1.7, v=2.0, r=0.08)
  movej([1.2956, -0.9524, 1.6, -0.4, 1.57, 0.0], a=1.7, v=2.0, r=0.08)
  movej([1.2917, -0.9488, 1.6, -0.4, 1.57, 0.0], a=1.7, v=2.0, r=0.08)
  movej([1.2878, -0.9452, 1.6, -0.4, 1.57, 0.0], a=1.7, v=2.0, r=0.08)
  movej([1.2839, -0.9418, 1.6, -0.4, 1.57, 0.0], a=1.7, v=2.0, r=0.08)
  movej([1.2801, -0.9384, 1.6, -0.4, 1.57, 0.0], a=1.7, v=2.0, r=0.08)
  movej([1.2763, -0.9352, 1.6, -0.4, 1.57, 0.0], a=1.7, v=2.0, r=0.08)
  movej([1.2725, -0.932, 1.6, -0.4, 1.57, 0.0], a=1.7, v=2.0, r=0.08)
  movej([1.2687, -0.9289, 1.6, -0.4, 1.57, 0.0], a=1.7, v=2.0, r=0.08)
  movej([1.2649, -0.926, 1.6, -0.4, 1.57, 0.0], a=1.7, v=2.0, r=0.08)
  movej([1.2612, -0.9231, 1.6, -0.4, 1.57, 0.0], a=1.7, v=2.0, r=0.08)
  movej([1.2574, -0.9203, 1.6, -0.4, 1.57, 0.0], a=1.7, v=2.0, r=0.08)
  movej([1.2537, -0.9177, 1.6, -0.4, 1.57, 0.0], a=1.7, v=2.0, r=0.08)
  movej([1.25, -0.9151, 1.6, -0.4, 1.57, 0.0], a=1.7, v=2.0, r=0.08)
  movej([1.2464, -0.9126, 1.6, -0.4, 1.57, 0.0], a=1.7, v=2.0, r=0.08)
  movej([1.2427, -0.9103, 1.6, -0.4, 1.57, 0.0], a=1.7, v=2.0, r=0.08)
  movej([1.2391, -0.908, 1.6, -0.4, 1.57, 0.0], a=1.7, v=2.0, r=0.08)
  movej([1.2355, -0.9058, 1.6, -0.4, 1.57, 0.0], a=1.7, v=2.0, r=0.08)
  movej([1.2319, -0.9038, 1.6, -0.4, 1.57, 0.0], a=1.7, v=2.0, r=0.08)
  movej([1.2283, -0.9018, 1.6, -0.4, 1.57, 0.0], a=1.7, v=2.0, r=0.08)
  movej([1.2248, -0.9, 1.6, -0.4, 1.57, 0.0], a=1.7, v=2.0, r=0.08)
  movej([1.2212, -0.8982, 1.6, -0.4, 1.57, 0.0], a=1.7, v=2.0, r=0.08)
  movej([1.2177, -0.8966, 1.6, -0.4, 1.57, 0.0], a=1.7, v=2.0, r=0.08)
  movej([1.2142, -0.8951, 1.6, -0.4, 1.57, 0.0], a=1.7, v=2.0, r=0.08)
  movej([1.2108, -0.8937, 1.6, -0.4, 1.57, 0.0], a=1.7, v=2.0, r=0.08)
  movej([1.2073, -0.8923, 1.6, -0.4, 1.57, 0.0], a=1.7, v=2.0, r=0.08)
  movej([1.2039, -0.8911, 1.6, -0.4, 1.57, 0.0], a=1.7, v=2.0, r=0.08)
  movej([1.2005, -0.89, 1.6, -0.4, 1.57, 0.0], a=1.7, v=2.0, r=0.08)
  movej([1.1972, -0.8891, 1.6, -0.4, 1.57, 0.0], a=1.7, v=2.0, r=0.08)
  movej([1.1938, -0.8882, 1.6, -0.4, 1.57, 0.0], a=1.7, v=2.0, r=0.08)
  movej([1.1905, -0.8874, 1.6, -0.4, 1.57, 0.0], a=1.7, v=2.0, r=0.08)
  movej([1.1872, -0.8867, 1.6, -0.4, 1.57, 0.0], a=1.7, v=2.0, r=0.08)
  movej([1.1839, -0.8862, 1.6, -0.4, 1.57, 0.0], a=1.7, v=2.0, r=0.08)
  movej([1.1807, -0.8857, 1.6, -0.4, 1.57, 0.0], a=1.7, v=2.0, r=0.08)
  movej([1.1774, -0.8854, 1.6, -0.4, 1.57, 0.0], a=1.7, v=2.0, r=0.08)
  movej([1.1742, -0.8851, 1.6, -0.4, 1.57, 0.0], a=1.7, v=2.0, r=0.08)
  movej([1.171, -0.885, 1.6, -0.4, 1.57, 0.0], a=1.7, v=2.0, r=0.08)
  movej([1.1679, -0.885, 1.6, -0.4, 1.57, 0.0], a=1.7, v=2.0, r=0.08)
  movej([1.1648, -0.8851, 1.6, -0.4, 1.57, 0.0], a=1.7, v=2.0, r=0.08)
  movej([1.1616, -0.8853, 1.6, -0.4, 1.57, 0.0], a=1.7, v=2.0, r=0.08)
  movej([1.1586, -0.8856, 1.6, -0.4, 1.57, 0.0], a=1.7, v=2.0, r=0.08)
  movej([1.1555, -0.886, 1.6, -0.4, 1.57, 0.0], a=1.7, v=2.0, r=0.08)
  movej([1.1525, -0.8866, 1.6, -0.4, 1.57, 0.0], a=1.7, v=2.0, r=0.08)
  movej([1.1495, -0.8872, 1.6, -0.4, 1.57, 0.0], a=1.7, v=2.0, r=0.08)
  movej([1.1465, -0.888, 1.6, -0.4, 1.57, 0.0], a=1.7, v=2.0, r=0.08)
  movej([1.1435, -0.8888, 1.6, -0.4, 1.57, 0.0], a=1.7, v=2.0, r=0.08)
  movej([1.1406, -0.8898, 1.6, -0.4, 1.57, 0.0], a=1.7, v=2.0, r=0.08)
  movej([1.1377, -0.8909, 1.6, -0.4, 1.57, 0.0], a=1.7, v=2.0, r=0.08)
  movej([1.1349, -0.892, 1.6, -0.4, 1.57, 0.0], a=1.7, v=2.0, r=0.08)
  movej([1.132, -0.8933, 1.6, -0.4, 1.57, 0.0], a=1.7, v=2.0, r=0.08)
  movej([1.1292, -0.8947, 1.6, -0.4, 1.57, 0.0], a=1.7, v=2.0, r=0.08)
  movej([1.1264, -0.8962, 1.6, -0.4, 1.57, 0.0], a=1.7, v=2.0, r=0.08)
  movej([1.1236, -0.8978, 1.6, -0.4, 1.57, 0.0], a=1.7, v=2.0, r=0.08)
  movej([1.1209, -0.8995, 1.6, -0.4, 1.57, 0.0], a=1.7, v=2.0, r=0.08)
  movej([1.1182, -0.9014, 1.6, -0.4, 1.57, 0.0], a=1.7, v=2.0, r=0.08)
  movej([1.1155, -0.9033, 1.6, -0.4, 1.57, 0.0], a=1.7, v=2.0, r=0.08)
  movej([1.1129, -0.9053, 1.6, -0.4, 1.57, 0.0], a=1.7, v=2.0, r=0.08)
  movej([1.1102, -0.9074, 1.6, -0.4, 1.57, 0.0], a=1.7, v=2.0, r=0.08)
  movej([1.1076, -0.9097, 1.6, -0.4, 1.57, 0.0], a=1.7, v=2.0, r=0.08)
  movej([1.1051, -0.912, 1.6, -0.4, 1.57, 0.0], a=1.7, v=2.0, r=0.08)
  movej([1.1025, -0.9145, 1.6, -0.4, 1.57, 0.0], a=1.7, v=2.0, r=0.08)
  movej([1.1, -0.917, 1.6, -0.4, 1.57, 0.0], a=1.7, v=2.0, r=0.08)
  movej([1.0975, -0.9197, 1.6, -0.4, 1.57, 0.0], a=1.7, v=2.0, r=0.08)
  movej([1.0951, -0.9224, 1.6, -0.4, 1.57, 0.0], a=1.7, v=2.0, r=0.08)
  movej([1.0927, -0.9252, 1.6, -0.4, 1.57, 0.0], a=1.7, v=2.0, r=0.08)
  movej([1.0903, -0.9282, 1.6, -0.4, 1.57, 0.0], a=1.7, v=2.0, r=0.08)
  movej([1.0879, -0.9312, 1.6, -0.4, 1.57, 0.0], a=1.7, v=2.0, r=0.08)
  movej([1.0856, -0.9344, 1.6, -0.4, 1.57, 0.0], a=1.7, v=2.0, r=0.08)
  movej([1.0833, -0.9376, 1.6, -0.4, 1.57, 0.0], a=1.7, v=2.0, r=0.08)
  movej([1.081, -0.9409, 1.6, -0.4, 1.57, 0.0], a=1.7, v=2.0, r=0.08)
  movej([1.0788, -0.9444, 1.6, -0.4, 1.57, 0.0], a=1.7, v=2.0, r=0.08)
  movej([1.0766, -0.9479, 1.6, -0.4, 1.57, 0.0], a=1.7, v=2.0, r=0.08)
  movej([1.0744, -0.9515, 1.6, -0.4, 1.57, 0.0], a=1.7, v=2.0, r=0.08)
  movej([1.0722, -0.9552, 1.6, -0.4, 1.57, 0.0], a=1.7, v=2.0, r=0.08)
  movej([1.0701, -0.959, 1.6, -0.4, 1.57, 0.0], a=1.7, v=2.0, r=0.08)
  movej([1.068, -0.9629, 1.6, -0.4, 1.57, 0.0], a=1.7, v=2.0, r=0.08)
  movej([1.066, -0.9669, 1.6, -0.4, 1.57, 0.0], a=1.7, v=2.0, r=0.08)
  movej([1.0639, -0.971, 1.6, -0.4, 1.57, 0.0], a=1.7, v=2.0, r=0.08)
  movej([1.0619, -0.9751, 1.6, -0.4, 1.57, 0.0], a=1.7, v=2.0, r=0.08)
  movej([1.06, -0.9794, 1.6, -0.4, 1.57, 0.0], a=1.7, v=2.0, r=0.08)
  movej([1.058, -0.9837, 1.6, -0.4, 1.57, 0.0], a=1.7, v=2.0, r=0.08)
  movej([1.0561, -0.9881, 1.6, -0.4, 1.57, 0.0], a=1.7, v=2.0, r=0.08)
  movej([1.0543, -0.9926, 1.6, -0.4, 1.57, 0.0], a=1.7, v=2.0, r=0.08)
  movej([1.0524, -0.9972, 1.6, -0.4, 1.57, 0.0], a=1.7, v=2.0, r=0.08)
  movej([1.0506, -1.0019, 1.6, -0.4, 1.57, 0.0], a=1.7, v=2.0, r=0.08)
  movej([1.0489, -1.0066, 1.6, -0.4, 1.57, 0.0], a=1.7, v=2.0, r=0.08)
  movej([1.0471, -1.0114, 1.6, -0.4, 1.57, 0.0], a=1.7, v=2.0, r=0.08)
  movej([1.0454, -1.0163, 1.6, -0.4, 1.57, 0.0], a=1.7, v=2.0, r=0.08)
  movej([1.0437, -1.0213, 1.6, -0.4, 1.57, 0.0], a=1.7, v=2.0, r=0.08)
  movej([1.0421, -1.0263, 1.6, -0.4, 1.57, 0.0], a=1.7, v=2.0, r=0.08)
  movej([1.0405, -1.0315, 1.6, -0.4, 1.57, 0.0], a=1.7, v=2.0, r=0.08)
  movej([1.0389, -1.0367, 1.6, -0.4, 1.57, 0.0], a=1.7, v=2.0, r=0.08)
  movej([1.0374, -1.0419, 1.6, -0.4, 1.57, 0.0], a=1.7, v=2.0, r=0.08)
  movej([1.0358, -1.0473, 1.6, -0.4, 1.57, 0.0], a=1.7, v=2.0, r=0.08)
  movej([1.0344, -1.0527, 1.6, -0.4, 1.57, 0.0], a=1.7, v=2.0, r=0.08)
  movej([1.0329, -1.0582, 1.6, -0.4, 1.57, 0.0], a=1.7, v=2.0, r=0.08)
  movej([1.0315, -1.0637, 1.6, -0.4, 1.57, 0.0], a=1.7, v=2.0, r=0.08)
  movej([1.0301, -1.0693, 1.6, -0.4, 1.57, 0.0], a=1.7, v=2.0, r=0.08)
  movej([1.0288, -1.075, 1.6, -0.4, 1.57, 0.0], a=1.7, v=2.0, r=0.08)
  movej([1.0275, -1.0807, 1.6, -0.4, 1.57, 0.0], a=1.7, v=2.0, r=0.08)
  movej([1.0262, -1.0865, 1.6, -0.4, 1.57, 0.0], a=1.7, v=2.0, r=0.08)
  movej([1.0249, -1.0924, 1.6, -0.4, 1.57, 0.0], a=1.7, v=2.0, r=0.08)
  movej([1.0237, -1.0983, 1.6, -0.4, 1.57, 0.0], a=1.7, v=2.0, r=0.08)
  movej([1.0226, -1.1042, 1.6, -0.4, 1.57, 0.0], a=1.7, v=2.0, r=0.08)
  movej([1.0214, -1.1103, 1.6, -0.4, 1.57, 0.0], a=1.7, v=2.0, r=0.08)
  movej([1.0203, -1.1163, 1.6, -0.4, 1.57, 0.0], a=1.7, v=2.0, r=0.08)
  movej([1.0192, -1.1225, 1.6, -0.4, 1.57, 0.0], a=1.7, v=2.0, r=0.08)
  movej([1.0182, -1.1287, 1.6, -0.4, 1.57, 0.0], a=1.7, v=2.0, r=0.08)
  movej([1.0172, -1.1349, 1.6, -0.4, 1.57, 0.0], a=1.7, v=2.0, r=0.08)
  movej([1.0162, -1.1412, 1.6, -0.4, 1.57, 0.0], a=1.7, v=2.0, r=0.08)
  movej([1.0153, -1.1475, 1.6, -0.4, 1.57, 0.0], a=1.7, v=2.0, r=0.08)
  movej([1.0144, -1.1538, 1.6, -0.4, 1.57, 0.0], a=1.7, v=2.0, r=0.08)
  movej([1.0135, -1.1602, 1.6, -0.4, 1.57, 0.0], a=1.7, v=2.0, r=0.08)
  movej([1.0126, -1.1667, 1.6, -0.4, 1.57, 0.0], a=1.7, v=2.0, r=0.08)
  movej([1.0118, -1.1732, 1.6, -0.4, 1.57, 0.0], a=1.7, v=2.0, r=0.08)
  movej([1.0111, -1.1797, 1.6, -0.4, 1.57, 0.0], a=1.7, v=2.0, r=0.08)
  movej([1.0103, -1.1863, 1.6, -0.4, 1.57, 0.0], a=1.7, v=2.0, r=0.08)
  movej([1.0096, -1.1929, 1.6, -0.4, 1.57, 0.0], a=1.7, v=2.0, r=0.08)
  movej([1.009, -1.1995, 1.6, -0.4, 1.57, 0.0], a=1.7, v=2.0, r=0.08)
  movej([1.0084, -1.2061, 1.6, -0.4, 1.57, 0.0], a=1.7, v=2.0, r=0.08)
  movej([1.0078, -1.2128, 1.6, -0.4, 1.57, 0.0], a=1.7, v=2.0, r=0.08)
  movej([1.0072, -1.2196, 1.6, -0.4, 1.57, 0.0], a=1.7, v=2.0, r=0.08)
  movej([1.0067, -1.2263, 1.6, -0.4, 1.57, 0.0], a=1.7, v=2.0, r=0.08)
  movej([1.0062, -1.2331, 1.6, -0.4, 1.57, 0.0], a=1.7, v=2.0, r=0.08)
  movej([1.0057, -1.2399, 1.6, -0.4, 1.57, 0.0], a=1.7, v=2.0, r=0.08)
  movej([1.0053, -1.2467, 1.6, -0.4, 1.57, 0.0], a=1.7, v=2.0, r=0.08)
  movej([1.0049, -1.2535, 1.6, -0.4, 1.57, 0.0], a=1.7, v=2.0, r=0.08)
  movej([1.0046, -1.2604, 1.6, -0.4, 1.57, 0.0], a=1.7, v=2.0, r=0.08)
  movej([1.0043, -1.2672, 1.6, -0.4, 1.57, 0.0], a=1.7, v=2.0, r=0.08)
  movej([1.004, -1.2741, 1.6, -0.4, 1.57, 0.0], a=1.7, v=2.0, r=0.08)
  movej([1.0037, -1.281, 1.6, -0.4, 1.57, 0.0], a=1.7, v=2.0, r=0.08)
  movej([1.0035, -1.2879, 1.6, -0.4, 1.57, 0.0], a=1.7, v=2.0, r=0.08)
  movej([1.0033, -1.2948, 1.6, -0.4, 1.57, 0.0], a=1.7, v=2.0, r=0.08)
  movej([1.0032, -1.3017, 1.6, -0.4, 1.57, 0.0], a=1.7, v=2.0, r=0.08)
  movej([1.0031, -1.3087, 1.6, -0.4, 1.57, 0.0], a=1.7, v=2.0, r=0.08)
  movej([1.003, -1.3156, 1.6, -0.4, 1.57, 0.0], a=1.7, v=2.0, r=0.08)
  movej([1.003, -1.3225, 1.6, -0.4, 1.57, 0.0], a=1.7, v=2.0, r=0.08)
  movej([1.003, -1.3295, 1.6, -0.4, 1.57, 0.0], a=1.7, v=2.0, r=0.08)
  movej([1.003, -1.3364, 1.6, -0.4, 1.57, 0.0], a=1.7, v=2.0, r=0.08)
  movej([1.0031, -1.3433, 1.6, -0.4, 1.57, 0.0], a=1.7, v=2.0, r=0.08)
  movej([1.0032, -1.3503, 1.6, -0.4, 1.57, 0.0], a=1.7, v=2.0, r=0.08)
  movej([1.0033, -1.3572, 1.6, -0.4, 1.57, 0.0], a=1.7, v=2.0, r=0.08)
  movej([1.0035, -1.3641, 1.6, -0.4, 1.57, 0.0], a=1.7, v=2.0, r=0.08)
  movej([1.0037, -1.371, 1.6, -0.4, 1.57, 0.0], a=1.7, v=2.0, r=0.08)
  movej([1.004, -1.3779, 1.6, -0.4, 1.57, 0.0], a=1.7, v=2.0, r=0.08)
  movej([1.0043, -1.3848, 1.6, -0.4, 1.57, 0.0], a=1.7, v=2.0, r=0.08)
  movej([1.0046, -1.3916, 1.6, -0.4, 1.57, 0.0], a=1.7, v=2.0, r=0.08)
  movej([1.0049, -1.3985, 1.6, -0.4, 1.57, 0.0], a=1.7, v=2.0, r=0.08)
  movej([1.0053, -1.4053, 1.6, -0.4, 1.57, 0.0], a=1.7, v=2.0, r=0.08)
  movej([1.0057, -1.4121, 1.6, -0.4, 1.57, 0.0], a=1.7, v=2.0, r=0.08)
  movej([1.0062, -1.4189, 1.6, -0.4, 1.57, 0.0], a=1.7, v=2.0, r=0.08)
  movej([1.0067, -1.4257, 1.6, -0.4, 1.57, 0.0], a=1.7, v=2.0, r=0.08)
  movej([1.0072, -1.4324, 1.6, -0.4, 1.57, 0.0], a=1.7, v=2.0, r=0.08)
  movej([1.0078, -1.4392, 1.6, -0.4, 1.57, 0.0], a=1.7, v=2.0, r=0.08)
  movej([1.0084, -1.4459, 1.6, -0.4, 1.57, 0.0], a=1.7, v=2.0, r=0.08)
  movej([1.009, -1.4525, 1.6, -0.4, 1.57, 0.0], a=1.7, v=2.0, r=0.08)
  movej([1.0096, -1.4591, 1.6, -0.4, 1.57, 0.0], a=1.7, v=2.0, r=0.08)
  movej([1.0103, -1.4657, 1.6, -0.4, 1.57, 0.0], a=1.7, v=2.0, r=0.08)
  movej([1.0111, -1.4723, 1.6, -0.4, 1.57, 0.0], a=1.7, v=2.0, r=0.08)
  movej([1.0118, -1.4788, 1.6, -0.4, 1.57, 0.0], a=1.7, v=2.0, r=0.08)
  movej([1.0126, -1.4853, 1.6, -0.4, 1.57, 0.0], a=1.7, v=2.0, r=0.08)
  movej([1.0135, -1.4918, 1.6, -0.4, 1.57, 0.0], a=1.7, v=2.0, r=0.08)
  movej([1.0144, -1.4982, 1.6, -0.4, 1.57, 0.0], a=1.7, v=2.0, r=0.08)
  movej([1.0153, -1.5045, 1.6, -0.4, 1.57, 0.0], a=1.7, v=2.0, r=0.08)
  movej([1.0162, -1.5108, 1.6, -0.4, 1.57, 0.0], a=1.7, v=2.0, r=0.08)
  movej([1.0172, -1.5171, 1.6, -0.4, 1.57, 0.0], a=1.7, v=2.0, r=0.08)
  movej([1.0182, -1.5233, 1.6, -0.4, 1.57, 0.0], a=1.7, v=2.0, r=0.08)
  movej([1.0192, -1.5295, 1.6, -0.4, 1.57, 0.0], a=1.7, v=2.0, r=0.08)
  movej([1.0203, -1.5357, 1.6, -0.4, 1.57, 0.0], a=1.7, v=2.0, r=0.08)
  movej([1.0214, -1.5417, 1.6, -0.4, 1.57, 0.0], a=1.7, v=2.0, r=0.08)
  movej([1.0226, -1.5478, 1.6, -0.4, 1.57, 0.0], a=1.7, v=2.0, r=0.08)
  movej([1.0237, -1.5537, 1.6, -0.4, 1.57, 0.0], a=1.7, v=2.0, r=0.08)
  movej([1.0249, -1.5596, 1.6, -0.4, 1.57, 0.0], a=1.7, v=2.0, r=0.08)
  movej([1.0262, -1.5655, 1.6, -0.4, 1.57, 0.0], a=1.7, v=2.0, r=0.08)
  movej([1.0275, -1.5713, 1.6, -0.4, 1.57, 0.0], a=1.7, v=2.0, r=0.08)
  movej([1.0288, -1.577, 1.6, -0.4, 1.57, 0.0], a=1.7, v=2.0, r=0.08)
  movej([1.0301, -1.5827, 1.6, -0.4, 1.57, 0.0], a=1.7, v=2.0, r=0.08)
  movej([1.0315, -1.5883, 1.6, -0.4, 1.57, 0.0], a=1.7, v=2.0, r=0.08)
  movej([1.0329, -1.5938, 1.6, -0.4, 1.57, 0.0], a=1.7, v=2.0, r=0.08)
  movej([1.0344, -1.5993, 1.6, -0.4, 1.57, 0.0], a=1.7, v=2.0, r=0.08)
  movej([1.0358, -1.6047, 1.6, -0.4, 1.57, 0.0], a=1.7, v=2.0, r=0.08)
  movej([1.0374, -1.6101, 1.6, -0.4, 1.57, 0.0], a=1.7, v=2.0, r=0.08)
  movej([1.0389, -1.6153, 1.6, -0.4, 1.57, 0.0], a=1.7, v=2.0, r=0.08)
  movej([1.0405, -1.6205, 1.6, -0.4, 1.57, 0.0], a=1.7, v=2.0, r=0.08)
  movej([1.0421, -1.6257, 1.6, -0.4, 1.57, 0.0], a=1.7, v=2.0, r=0.08)
  movej([1.0437, -1.6307, 1.6, -0.4, 1.57, 0.0], a=1.7, v=2.0, r=0.08)
  movej([1.0454, -1.6357, 1.6, -0.4, 1.57, 0.0], a=1.7, v=2.0, r=0.08)
  movej([1.0471, -1.6406, 1.6, -0.4, 1.57, 0.0], a=1.7, v=2.0, r=0.08)
  movej([1.0489, -1.6454, 1.6, -0.4, 1.57, 0.0], a=1.7, v=2.0, r=0.08)
  movej([1.0506, -1.6501, 1.6, -0.4, 1.57, 0.0], a=1.7, v=2.0, r=0.08)
  movej([1.0524, -1.6548, 1.6, -0.4, 1.57, 0.0], a=1.7, v=2.0, r=0.08)
  movej([1.0543, -1.6594, 1.6, -0.4, 1.57, 0.0], a=1.7, v=2.0, r=0.08)
  movej([1.0561, -1.6639, 1.6, -0.4, 1.57, 0.0], a=1.7, v=2.0, r=0.08)
  movej([1.058, -1.6683, 1.6, -0.4, 1.57, 0.0], a=1.7, v=2.0, r=0.08)
  movej([1.06, -1.6726, 1.6, -0.4, 1.57, 0.0], a=1.7, v=2.0, r=0.08)
  movej([1.0619, -1.6769, 1.6, -0.4, 1.57, 0.0], a=1.7, v=2.0, r=0.08)
  movej([1.0639, -1.681, 1.6, -0.4, 1.57, 0.0], a=1.7, v=2.0, r=0.08)
  movej([1.066, -1.6851, 1.6, -0.4, 1.57, 0.0], a=1.7, v=2.0, r=0.08)
  movej([1.068, -1.6891, 1.6, -0.4, 1.57, 0.0], a=1.7, v=2.0, r=0.08)
  movej([1.0701, -1.693, 1.6, -0.4, 1.57, 0.0], a=1.7, v=2.0, r=0.08)
  movej([1.0722, -1.6968, 1.6, -0.4, 1.57, 0.0], a=1.7, v=2.0, r=0.08)
  movej([1.0744, -1.7005, 1.6, -0.4, 1.57, 0.0], a=1.7, v=2.0, r=0.08)
  movej([1.0766, -1.7041, 1.6, -0.4, 1.57, 0.0], a=1.7, v=2.0, r=0.08)
  movej([1.0788, -1.7076, 1.6, -0.4, 1.57, 0.0], a=1.7, v=2.0, r=0.08)
  movej([1.081, -1.7111, 1.6, -0.4, 1.57, 0.0], a=1.7, v=2.0, r=0.08)
  movej([1.0833, -1.7144, 1.6, -0.4, 1.57, 0.0], a=1.7, v=2.0, r=0.08)
  movej([1.0856, -1.7176, 1.6, -0.4, 1.57, 0.0], a=1.7, v=2.0, r=0.08)
  movej([1.0879, -1.7208, 1.6, -0.4, 1.57, 0.0], a=1.7, v=2.0, r=0.08)
  movej([1.0903, -1.7238, 1.6, -0.4, 1.57, 0.0], a=1.7, v=2.0, r=0.08)
  movej([1.0927, -1.7268, 1.6, -0.4, 1.57, 0.0], a=1.7, v=2.0, r=0.08)
  movej([1.0951, -1.7296, 1.6, -0.4, 1.57, 0.0], a=1.7, v=2.0, r=0.08)
  movej([1.0975, -1.7323, 1.6, -0.4, 1.57, 0.0], a=1.7, v=2.0, r=0.08)
  movej([1.1, -1.735, 1.6, -0.4, 1.57, 0.0], a=1.7, v=2.0, r=0.08)
  movej([1.1025, -1.7375, 1.6, -0.4, 1.57, 0.0], a=1.7, v=2.0, r=0.08)
  movej([1.1051, -1.74, 1.6, -0.4, 1.57, 0.0], a=1.7, v=2.0, r=0.08)
  movej([1.1076, -1.7423, 1.6, -0.4, 1.57, 0.0], a=1.7, v=2.0, r=0.08)
  movej([1.1102, -1.7446, 1.6, -0.4, 1.57, 0.0], a=1.7, v=2.0, r=0.08)
  movej([1.1129, -1.7467, 1.6, -0.4, 1.57, 0.0], a=1.7, v=2.0, r=0.08)
  movej([1.1155, -1.7487, 1.6, -0.4, 1.57, 0.0], a=1.7, v=2.0, r=0.08)
  movej([1.1182, -1.7506, 1.6, -0.4, 1.57, 0.0], a=1.7, v=2.0, r=0.08)
  movej([1.1209, -1.7525, 1.6, -0.4, 1.57, 0.0], a=1.7, v=2.0, r=0.08)
  movej([1.1236, -1.7542, 1.6, -0.4, 1.57, 0.0], a=1.7, v=2.0, r=0.08)
  movej([1.1264, -1.7558, 1.6, -0.4, 1.57, 0.0], a=1.7, v=2.0, r=0.08)
  movej([1.1292, -1.7573, 1.6, -0.4, 1.57, 0.0], a=1.7, v=2.0, r=0.08)
  movej([1.132, -1.7587, 1.6, -0.4, 1.57, 0.0], a=1.7, v=2.0, r=0.08)
  movej([1.1349, -1.76, 1.6, -0.4, 1.57, 0.0], a=1.7, v=2.0, r=0.08)
  movej([1.1377, -1.7611, 1.6, -0.4, 1.57, 0.0], a=1.7, v=2.0, r=0.08)
  movej([1.1406, -1.7622, 1.6, -0.4, 1.57, 0.0], a=1.7, v=2.0, r=0.08)
  movej([1.1435, -1.7632, 1.6, -0.4, 1.57, 0.0], a=1.7, v=2.0, r=0.08)
  movej([1.1465, -1.764, 1.6, -0.4, 1.57, 0.0], a=1.7, v=2.0, r=0.08)
  movej([1.1495, -1.7648, 1.6, -0.4, 1.57, 0.0], a=1.7, v=2.0, r=0.08)
  movej([1.1525, -1.7654, 1.6, -0.4, 1.57, 0.0], a=1.7, v=2.0, r=0.08)
  movej([1.1555, -1.766, 1.6, -0.4, 1.57, 0.0], a=1.7, v=2.0, r=0.08)
  movej([1.1586, -1.7664, 1.6, -0.4, 1.57, 0.0], a=1.7, v=2.0, r=0.08)
  movej([1.1616, -1.7667, 1.6, -0.4, 1.57, 0.0], a=1.7, v=2.0, r=0.08)
  movej([1.1648, -1.7669, 1.6, -0.4, 1.57, 0.0], a=1.7, v=2.0, r=0.08)
  movej([1.1679, -1.767, 1.6, -0.4, 1.57, 0.0], a=1.7, v=2.0, r=0.08)
  movej([1.171, -1.767, 1.6, -0.4, 1.57, 0.0], a=1.7, v=2.0, r=0.08)
  movej([1.1742, -1.7669, 1.6, -0.4, 1.57, 0.0], a=1.7, v=2.0, r=0.08)
  movej([1.1774, -1.7666, 1.6, -0.4, 1.57, 0.0], a=1.7, v=2.0, r=0.08)
  movej([1.1807, -1.7663, 1.6, -0.4, 1.57, 0.0], a=1.7, v=2.0, r=0.08)
  movej([1.1839, -1.7658, 1.6, -0.4, 1.57, 0.0], a=1.7, v=2.0, r=0.08)
  movej([1.1872, -1.7653, 1.6, -0.4, 1.57, 0.0], a=1.7, v=2.0, r=0.08)
  movej([1.1905, -1.7646, 1.6, -0.4, 1.57, 0.0], a=1.7, v=2.0, r=0.08)
  movej([1.1938, -1.7638, 1.6, -0.4, 1.57, 0.0], a=1.7, v=2.0, r=0.08)
  movej([1.1972, -1.7629, 1.6, -0.4, 1.57, 0.0], a=1.7, v=2.0, r=0.08)
  movej([1.2005, -1.762, 1.6, -0.4, 1.57, 0.0], a=1.7, v=2.0, r=0.08)
  movej([1.2039, -1.7609, 1.6, -0.4, 1.57, 0.0], a=1.7, v=2.0, r=0.08)
  movej([1.2073, -1.7597, 1.6, -0.4, 1.57, 0.0], a=1.7, v=2.0, r=0.08)
  movej([1.2108, -1.7583, 1.6, -0.4, 1.57, 0.0], a=1.7, v=2.0, r=0.08)
  movej([1.2142, -1.7569, 1.6, -0.4, 1.57, 0.0], a=1.7, v=2.0, r=0.08)
  movej([1.2177, -1.7554, 1.6, -0.4, 1.57, 0.0], a=1.7, v=2.0, r=0.08)
  movej([1.2212, -1.7538, 1.6, -0.4, 1.57, 0.0], a=1.7, v=2.0, r=0.08)
  movej([1.2248, -1.752, 1.6, -0.4, 1.57, 0.0], a=1.7, v=2.0, r=0.08)
  movej([1.2283, -1.7502, 1.6, -0.4, 1.57, 0.0], a=1.7, v=2.0, r=0.08)
  movej([1.2319, -1.7482, 1.6, -0.4, 1.57, 0.0], a=1.7, v=2.0, r=0.08)
  movej([1.2355, -1.7462, 1.6, -0.4, 1.57, 0.0], a=1.7, v=2.0, r=0.08)
  movej([1.2391, -1.744, 1.6, -0.4, 1.57, 0.0], a=1.7, v=2.0, r=0.08)
  movej([1.2427, -1.7417, 1.6, -0.4, 1.57, 0.0], a=1.7, v=2.0, r=0.08)
  movej([1.2464, -1.7394, 1.6, -0.4, 1.57, 0.0], a=1.7, v=2.0, r=0.08)
  movej([1.25, -1.7369, 1.6, -0.4, 1.57, 0.0], a=1.7, v=2.0, r=0.08)
  movej([1.2537, -1.7343, 1.6, -0.4, 1.57, 0.0], a=1.7, v=2.0, r=0.08)
  movej([1.2574, -1.7317, 1.6, -0.4, 1.57, 0.0], a=1.7, v=2.0, r=0.08)
  movej([1.2612, -1.7289, 1.6, -0.4, 1.57, 0.0], a=1.7, v=2.0, r=0.08)
  movej([1.2649, -1.726, 1.6, -0.4, 1.57, 0.0], a=1.7, v=2.0, r=0.08)
  movej([1.2687, -1.7231, 1.6, -0.4, 1.57, 0.0], a=1.7, v=2.0, r=0.08)
  movej([1.2725, -1.72, 1.6, -0.4, 1.57, 0.0], a=1.7, v=2.0, r=0.08)
  movej([1.2763, -1.7168, 1.6, -0.4, 1.57, 0.0], a=1.7, v=2.0, r=0.08)
  movej([1.2801, -1.7136, 1.6, -0.4, 1.57, 0.0], a=1.7, v=2.0, r=0.08)
  movej([1.2839, -1.7102, 1.6, -0.4, 1.57, 0.0], a=1.7, v=2.0, r=0.08)
  movej([1.2878, -1.7068, 1.6, -0.4, 1.57, 0.0], a=1.7, v=2.0, r=0.08)
  movej([1.2917, -1.7032, 1.6, -0.4, 1.57, 0.0], a=1.7, v=2.0, r=0.08)
  movej([1.2956, -1.6996, 1.6, -0.4, 1.57, 0.0], a=1.7, v=2.0, r=0.08)
  movej([1.2995, -1.6958, 1.6, -0.4, 1.57, 0.0], a=1.7, v=2.0, r=0.08)
  movej([1.3034, -1.692, 1.6, -0.4, 1.57, 0.0], a=1.7, v=2.0, r=0.08)
  movej([1.3073, -1.6881, 1.6, -0.4, 1.57, 0.0], a=1.7, v=2.0, r=0.08)
  movej([1.3113, -1.6841, 1.6, -0.4, 1.57, 0.0], a=1.7, v=2.0, r=0.08)
  movej([1.3153, -1.68, 1.6, -0.4, 1.57, 0.0], a=1.7, v=2.0, r=0.08)
  movej([1.3193, -1.6758, 1.6, -0.4, 1.57, 0.0], a=1.7, v=2.0, r=0.08)
  movej([1.3233, -1.6716, 1.6, -0.4, 1.57, 0.0], a=1.7, v=2.0, r=0.08)
  movej([1.3273, -1.6672, 1.6, -0.4, 1.57, 0.0], a=1.7, v=2.0, r=0.08)
  movej([1.3313, -1.6628, 1.6, -0.4, 1.57, 0.0], a=1.7, v=2.0, r=0.08)
  movej([1.3354, -1.6583, 1.6, -0.4, 1.57, 0.0], a=1.7, v=2.0, r=0.08)
  movej([1.3394, -1.6537, 1.6, -0.4, 1.57, 0.0], a=1.7, v=2.0, r=0.08)
  movej([1.3435, -1.649, 1.6, -0.4, 1.57, 0.0], a=1.7, v=2.0, r=0.08)
  movej([1.3476, -1.6442, 1.6, -0.4, 1.57, 0.0], a=1.7, v=2.0, r=0.08)
  movej([1.3517, -1.6394, 1.6, -0.4, 1.57, 0.0], a=1.7, v=2.0, r=0.08)
  movej([1.3558, -1.6344, 1.6, -0.4, 1.57, 0.0], a=1.7, v=2.0, r=0.08)
  movej([1.36, -1.6294, 1.6, -0.4, 1.57, 0.0], a=1.7, v=2.0, r=0.08)
  movej([1.3641, -1.6244, 1.6, -0.4, 1.57, 0.0], a=1.7, v=2.0, r=0.08)
  movej([1.3683, -1.6192, 1.6, -0.4, 1.57, 0.0], a=1.7, v=2.0, r=0.08)
  movej([1.3725, -1.614, 1.6, -0.4, 1.57, 0.0], a=1.7, v=2.0, r=0.08)
  movej([1.3767, -1.6087, 1.6, -0.4, 1.57, 0.0], a=1.7, v=2.0, r=0.08)
  movej([1.3809, -1.6034, 1.6, -0.4, 1.57, 0.0], a=1.7, v=2.0, r=0.08)
  movej([1.3851, -1.5979, 1.6, -0.4, 1.57, 0.0], a=1.7, v=2.0, r=0.08)
  movej([1.3893, -1.5925, 1.6, -0.4, 1.57, 0.0], a=1.7, v=2.0, r=0.08)
  movej([1.3935, -1.5869, 1.6, -0.4, 1.57, 0.0], a=1.7, v=2.0, r=0.08)
  movej([1.3978, -1.5813, 1.6, -0.4, 1.57, 0.0], a=1.7, v=2.0, r=0.08)
  movej([1.402, -1.5756, 1.6, -0.4, 1.57, 0.0], a=1.7, v=2.0, r=0.08)
  movej([1.4063, -1.5698, 1.6, -0.4, 1.57, 0.0], a=1.7, v=2.0, r=0.08)
  movej([1.4105, -1.564, 1.6, -0.4, 1.57, 0.0], a=1.7, v=2.0, r=0.08)
  movej([1.4148, -1.5582, 1.6, -0.4, 1.57, 0.0], a=1.7, v=2.0, r=0.08)
  movej([1.4191, -1.5522, 1.6, -0.4, 1.57, 0.0], a=1.7, v=2.0, r=0.08)
  movej([1.4234, -1.5463, 1.6, -0.4, 1.57, 0.0], a=1.7, v=2.0, r=0.08)
  movej([1.4277, -1.5402, 1.6, -0.4, 1.57, 0.0], a=1.7, v=2.0, r=0.08)
  movej([1.4321, -1.5341, 1.6, -0.4, 1.57, 0.0], a=1.7, v=2.0, r=0.08)
  movej([1.4364, -1.528, 1.6, -0.4, 1.57, 0.0], a=1.7, v=2.0, r=0.08)
  movej([1.4407, -1.5218, 1.6, -0.4, 1.57, 0.0], a=1.7, v=2.0, r=0.08)
  movej([1.4451, -1.5156, 1.6, -0.4, 1.57, 0.0], a=1.7, v=2.0, r=0.08)
  movej([1.4494, -1.5093, 1.6, -0.4, 1.57, 0.0], a=1.7, v=2.0, r=0.08)
  movej([1.4538, -1.5029, 1.6, -0.4, 1.57, 0.0], a=1.7, v=2.0, r=0.08)
  movej([1.4582, -1.4966, 1.6, -0.4, 1.57, 0.0], a=1.7, v=2.0, r=0.08)
  movej([1.4625, -1.4901, 1.6, -0.4, 1.57, 0.0], a=1.7, v=2.0, r=0.08)
  movej([1.4669, -1.4837, 1.6, -0.4, 1.57, 0.0], a=1.7, v=2.0, r=0.08)
  movej([1.4713, -1.4772, 1.6, -0.4, 1.57, 0.0], a=1.7, v=2.0, r=0.08)
  movej([1.4757, -1.4707, 1.6, -0.4, 1.57, 0.0], a=1.7, v=2.0, r=0.08)
  movej([1.4801, -1.4641, 1.6, -0.4, 1.57, 0.0], a=1.7, v=2.0, r=0.08)
  movej([1.4845, -1.4575, 1.6, -0.4, 1.57, 0.0], a=1.7, v=2.0, r=0.08)
  movej([1.4889, -1.4508, 1.6, -0.4, 1.57, 0.0], a=1.7, v=2.0, r=0.08)
  movej([1.4933, -1.4442, 1.6, -0.4, 1.57, 0.0], a=1.7, v=2.0, r=0.08)
  movej([1.4977, -1.4375, 1.6, -0.4, 1.57, 0.0], a=1.7, v=2.0, r=0.08)
  movej([1.5022, -1.4308, 1.6, -0.4, 1.57, 0.0], a=1.7, v=2.0, r=0.08)
  movej([1.5066, -1.424, 1.6, -0.4, 1.57, 0.0], a=1.7, v=2.0, r=0.08)
  movej([1.511, -1.4172, 1.6, -0.4, 1.57, 0.0], a=1.7, v=2.0, r=0.08)
  movej([1.5155, -1.4104, 1.6, -0.4, 1.57, 0.0], a=1.7, v=2.0, r=0.08)
  movej([1.5199, -1.4036, 1.6, -0.4, 1.57, 0.0], a=1.7, v=2.0, r=0.08)
  movej([1.5243, -1.3968, 1.6, -0.4, 1.57, 0.0], a=1.7, v=2.0, r=0.08)
  movej([1.5288, -1.3899, 1.6, -0.4, 1.57, 0.0], a=1.7, v=2.0, r=0.08)
  movej([1.5332, -1.3831, 1.6, -0.4, 1.57, 0.0], a=1.7, v=2.0, r=0.08)
  movej([1.5377, -1.3762, 1.6, -0.4, 1.57, 0.0], a=1.7, v=2.0, r=0.08)
  movej([1.5421, -1.3693, 1.6, -0.4, 1.57, 0.0], a=1.7, v=2.0, r=0.08)
  movej([1.5466, -1.3624, 1.6, -0.4, 1.57, 0.0], a=1.7, v=2.0, r=0.08)
  movej([1.5511, -1.3555, 1.6, -0.4, 1.57, 0.0], a=1.7, v=2.0, r=0.08)
  movej([1.5555, -1.3485, 1.6, -0.4, 1.57, 0.0], a=1.7, v=2.0, r=0.08)
  movej([1.56, -1.3416, 1.6, -0.4, 1.57, 0.0], a=1.7, v=2.0, r=0.08)
  movej([1.5644, -1.3347, 1.6, -0.4, 1.57, 0.0], a=1.7, v=2.0, r=0.08)
  movej([1.5689, -1.3277, 1.6, -0.4, 1.57, 0.0], a=1.7, v=2.0, r=0.08)
  movej([1.5733, -1.3208, 1.6, -0.4, 1.57, 0.0], a=1.7, v=2.0, r=0.08)
  movej([1.5778, -1.3139, 1.6, -0.4, 1.57, 0.0], a=1.7, v=2.0, r=0.08)
  movej([1.5823, -1.3069, 1.6, -0.4, 1.57, 0.0], a=1.7, v=2.0, r=0.08)
  movej([1.5867, -1.3, 1.6, -0.4, 1.57, 0.0], a=1.7, v=2.0, r=0.08)
  movej([1.5912, -1.2931, 1.6, -0.4, 1.57, 0.0], a=1.7, v=2.0, r=0.08)
  movej([1.5956, -1.2862, 1.6, -0.4, 1.57, 0.0], a=1.7, v=2.0, r=0.08)
